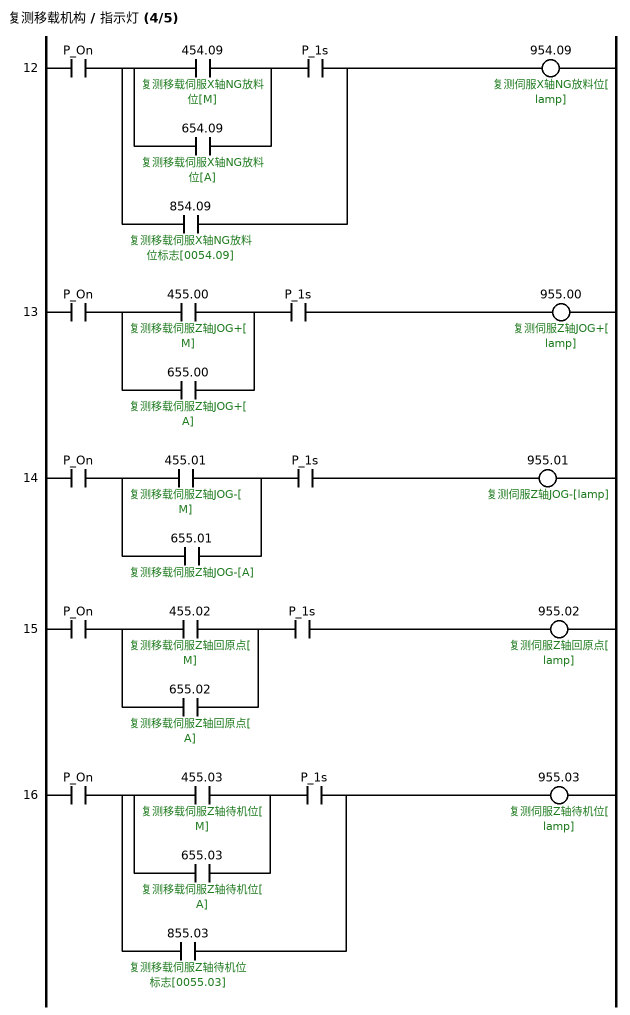
; [picture p576: 复测移载机构 / 指示灯, rungs 12-16]
; rung 12
LD P_On
LD 454.09  ; 复测移载伺服X轴NG放料位[M]
OR 654.09  ; 复测移载伺服X轴NG放料位[A]
AND P_1s
OR 854.09  ; 复测移载伺服X轴NG放料位标志[0054.09]
ANDLD
OUT 954.09  ; 复测伺服X轴NG放料位[lamp]
; rung 13
LD P_On
LD 455.00  ; 复测移载伺服Z轴JOG+[M]
OR 655.00  ; 复测移载伺服Z轴JOG+[A]
ANDLD
AND P_1s
OUT 955.00  ; 复测伺服Z轴JOG+[lamp]
; rung 14
LD P_On
LD 455.01  ; 复测移载伺服Z轴JOG-[M]
OR 655.01  ; 复测移载伺服Z轴JOG-[A]
ANDLD
AND P_1s
OUT 955.01  ; 复测伺服Z轴JOG-[lamp]
; rung 15
LD P_On
LD 455.02  ; 复测移载伺服Z轴回原点[M]
OR 655.02  ; 复测移载伺服Z轴回原点[A]
ANDLD
AND P_1s
OUT 955.02  ; 复测伺服Z轴回原点[lamp]
; rung 16
LD P_On
LD 455.03  ; 复测移载伺服Z轴待机位[M]
OR 655.03  ; 复测移载伺服Z轴待机位[A]
AND P_1s
OR 855.03  ; 复测移载伺服Z轴待机位标志[0055.03]
ANDLD
OUT 955.03  ; 复测伺服Z轴待机位[lamp]

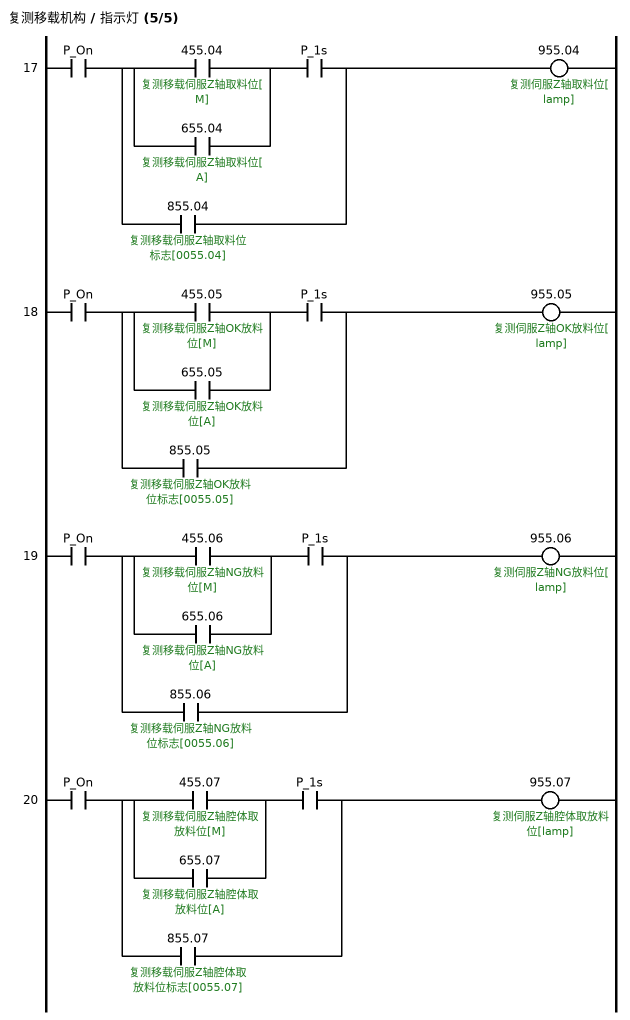
; rung 17
LD P_On
LD 455.04  ; 复测移载伺服Z轴取料位[M]
OR 655.04  ; 复测移载伺服Z轴取料位[A]
AND P_1s
OR 855.04  ; 复测移载伺服Z轴取料位标志[0055.04]
ANDLD
OUT 955.04  ; 复测伺服Z轴取料位[lamp]
; rung 18
LD P_On
LD 455.05  ; 复测移载伺服Z轴OK放料位[M]
OR 655.05  ; 复测移载伺服Z轴OK放料位[A]
AND P_1s
OR 855.05  ; 复测移载伺服Z轴OK放料位标志[0055.05]
ANDLD
OUT 955.05  ; 复测伺服Z轴OK放料位[lamp]
; rung 19
LD P_On
LD 455.06  ; 复测移载伺服Z轴NG放料位[M]
OR 655.06  ; 复测移载伺服Z轴NG放料位[A]
AND P_1s
OR 855.06  ; 复测移载伺服Z轴NG放料位标志[0055.06]
ANDLD
OUT 955.06  ; 复测伺服Z轴NG放料位[lamp]
; rung 20
LD P_On
LD 455.07  ; 复测移载伺服Z轴腔体取放料位[M]
OR 655.07  ; 复测移载伺服Z轴腔体取放料位[A]
AND P_1s
OR 855.07  ; 复测移载伺服Z轴腔体取放料位标志[0055.07]
ANDLD
OUT 955.07  ; 复测伺服Z轴腔体取放料位[lamp]

### Section 外部输出

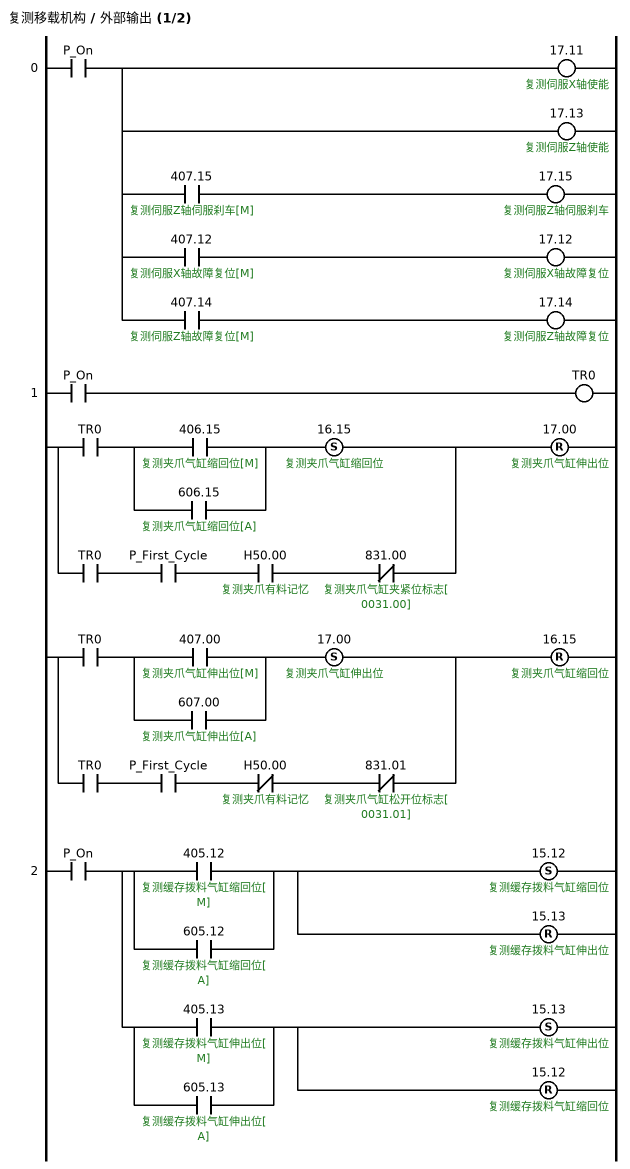
; rung 0
LD P_On
OUT TR0
OUT 17.11  ; 复测伺服X轴使能
OUT 17.13  ; 复测伺服Z轴使能
AND 407.15  ; 复测伺服Z轴伺服刹车[M]
OUT 17.15  ; 复测伺服Z轴伺服刹车
LD TR0
AND 407.12  ; 复测伺服X轴故障复位[M]
OUT 17.12  ; 复测伺服X轴故障复位
LD TR0
AND 407.14  ; 复测伺服Z轴故障复位[M]
OUT 17.14  ; 复测伺服Z轴故障复位
; rung 1
LD P_On
OUT TR0
LD 406.15  ; 复测夹爪气缸缩回位[M]
OR 606.15  ; 复测夹爪气缸缩回位[A]
ANDLD
SET 16.15  ; 复测夹爪气缸缩回位
LD TR0
AND P_First_Cycle
AND H50.00  ; 复测夹爪有料记忆
ANDNOT 831.00  ; 复测夹爪气缸夹紧位标志[0031.00]
ORLD
RSET 17.00  ; 复测夹爪气缸伸出位
LD TR0
LD 407.00  ; 复测夹爪气缸伸出位[M]
OR 607.00  ; 复测夹爪气缸伸出位[A]
ANDLD
SET 17.00  ; 复测夹爪气缸伸出位
LD TR0
AND P_First_Cycle
ANDNOT H50.00  ; 复测夹爪有料记忆
ANDNOT 831.01  ; 复测夹爪气缸松开位标志[0031.01]
ORLD
RSET 16.15  ; 复测夹爪气缸缩回位
; rung 2
LD P_On
OUT TR0
LD 405.12  ; 复测缓存拨料气缸缩回位[M]
OR 605.12  ; 复测缓存拨料气缸缩回位[A]
ANDLD
SET 15.12  ; 复测缓存拨料气缸缩回位
RSET 15.13  ; 复测缓存拨料气缸伸出位
LD TR0
LD 405.13  ; 复测缓存拨料气缸伸出位[M]
OR 605.13  ; 复测缓存拨料气缸伸出位[A]
ANDLD
SET 15.13  ; 复测缓存拨料气缸伸出位
RSET 15.12  ; 复测缓存拨料气缸缩回位

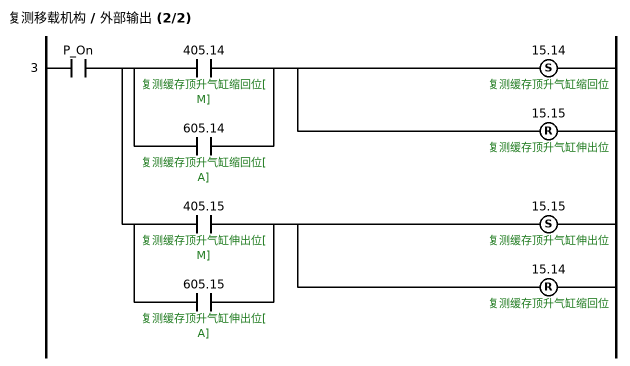
; rung 3
LD P_On
OUT TR0
LD 405.14  ; 复测缓存顶升气缸缩回位[M]
OR 605.14  ; 复测缓存顶升气缸缩回位[A]
ANDLD
SET 15.14  ; 复测缓存顶升气缸缩回位
RSET 15.15  ; 复测缓存顶升气缸伸出位
LD TR0
LD 405.15  ; 复测缓存顶升气缸伸出位[M]
OR 605.15  ; 复测缓存顶升气缸伸出位[A]
ANDLD
SET 15.15  ; 复测缓存顶升气缸伸出位
RSET 15.14  ; 复测缓存顶升气缸缩回位

### Section END
; rung 0
END(001)

## Program 复测腔体机构 (cyclic task 7)

### Section Main

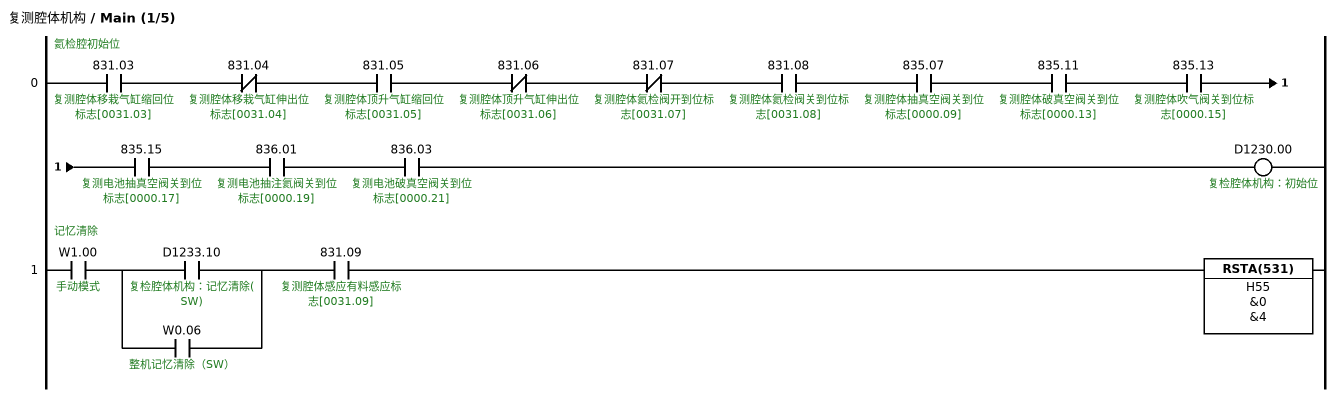
; rung 0: 氦检腔初始位
LD 831.03  ; 复测腔体移栽气缸缩回位标志[0031.03]
ANDNOT 831.04  ; 复测腔体移栽气缸伸出位标志[0031.04]
AND 831.05  ; 复测腔体顶升气缸缩回位标志[0031.05]
ANDNOT 831.06  ; 复测腔体顶升气缸伸出位标志[0031.06]
ANDNOT 831.07  ; 复测腔体氦检阀开到位标志[0031.07]
AND 831.08  ; 复测腔体氦检阀关到位标志[0031.08]
AND 835.07  ; 复测腔体抽真空阀关到位标志[0000.09]
AND 835.11  ; 复测腔体破真空阀关到位标志[0000.13]
AND 835.13  ; 复测腔体吹气阀关到位标志[0000.15]
AND 835.15  ; 复测电池抽真空阀关到位标志[0000.17]
AND 836.01  ; 复测电池抽注氦阀关到位标志[0000.19]
AND 836.03  ; 复测电池破真空阀关到位标志[0000.21]
OUT D1230.00  ; 复检腔体机构：初始位
; rung 1: 记忆清除
LD W1.00  ; 手动模式
LD D1233.10  ; 复检腔体机构：记忆清除(SW)
OR W0.06  ; 整机记忆清除（SW）
ANDLD
AND 831.09  ; 复测腔体感应有料感应标志[0031.09]
RSTA(531) H55 &0 &4

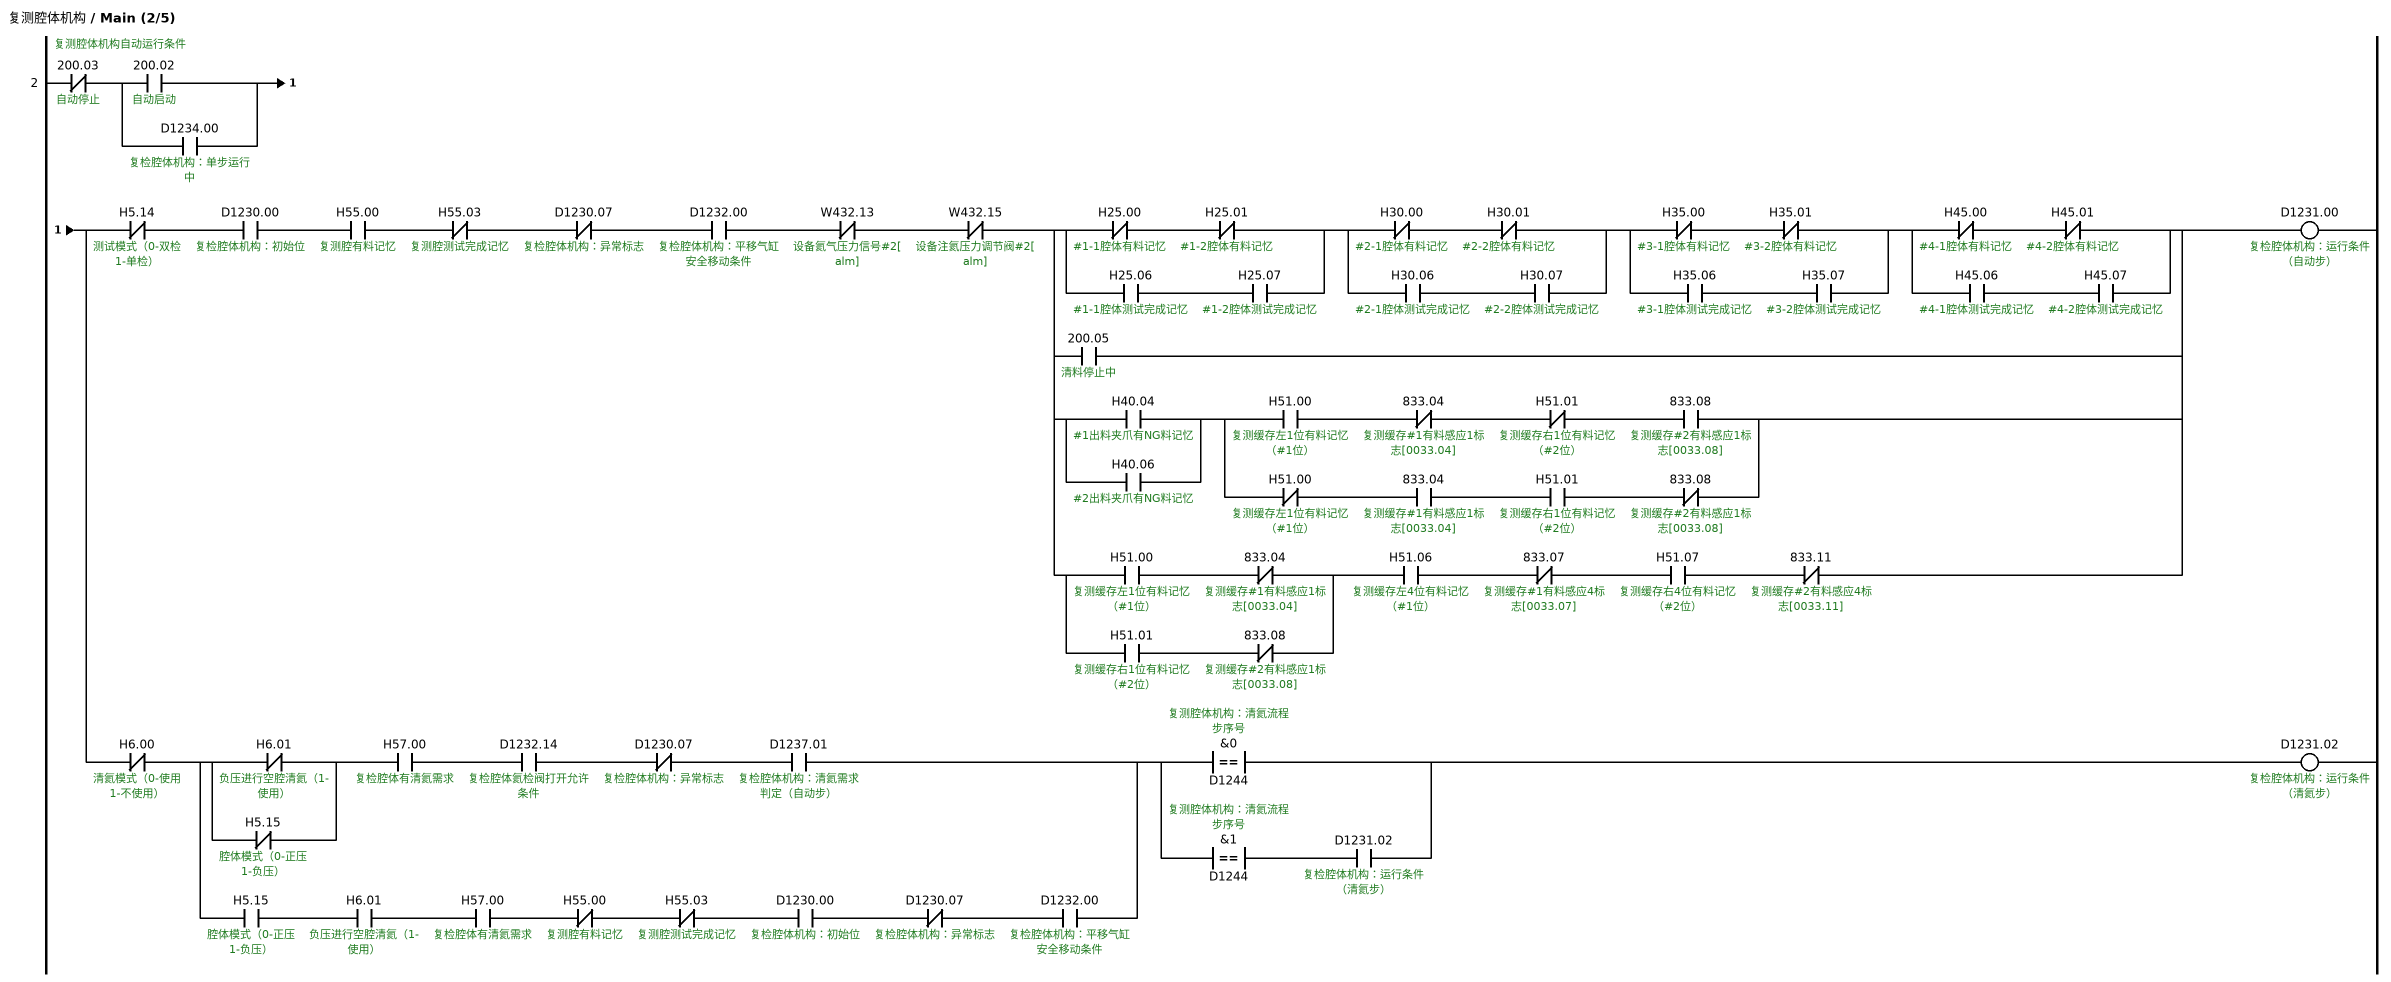
; rung 2: 复测腔体机构自动运行条件
LDNOT 200.03  ; 自动停止
LD 200.02  ; 自动启动
OR D1234.00  ; 复检腔体机构：单步运行中
ANDLD
OUT TR0
ANDNOT H5.14  ; 测试模式（0-双检 1-单检）
AND D1230.00  ; 复检腔体机构：初始位
AND H55.00  ; 复测腔有料记忆
ANDNOT H55.03  ; 复测腔测试完成记忆
ANDNOT D1230.07  ; 复检腔体机构：异常标志
AND D1232.00  ; 复检腔体机构：平移气缸安全移动条件
ANDNOT W432.13  ; 设备氦气压力信号#2[alm]
ANDNOT W432.15  ; 设备注氦压力调节阀#2[alm]
LDNOT H25.00  ; #1-1腔体有料记忆
ANDNOT H25.01  ; #1-2腔体有料记忆
LD H25.06  ; #1-1腔体测试完成记忆
AND H25.07  ; #1-2腔体测试完成记忆
ORLD
LDNOT H30.00  ; #2-1腔体有料记忆
ANDNOT H30.01  ; #2-2腔体有料记忆
LD H30.06  ; #2-1腔体测试完成记忆
AND H30.07  ; #2-2腔体测试完成记忆
ORLD
ANDLD
LDNOT H35.00  ; #3-1腔体有料记忆
ANDNOT H35.01  ; #3-2腔体有料记忆
LD H35.06  ; #3-1腔体测试完成记忆
AND H35.07  ; #3-2腔体测试完成记忆
ORLD
ANDLD
LDNOT H45.00  ; #4-1腔体有料记忆
ANDNOT H45.01  ; #4-2腔体有料记忆
LD H45.06  ; #4-1腔体测试完成记忆
AND H45.07  ; #4-2腔体测试完成记忆
ORLD
ANDLD
OR 200.05  ; 清料停止中
LD H40.04  ; #1出料夹爪有NG料记忆
OR H40.06  ; #2出料夹爪有NG料记忆
LD H51.00  ; 复测缓存左1位有料记忆（#1位）  // 缓存第一位出现单料是需直接清掉，防止下次待测料无法进行单个放料
ANDNOT 833.04  ; 复测缓存#1有料感应1标志[0033.04]
ANDNOT H51.01  ; 复测缓存右1位有料记忆（#2位）
AND 833.08  ; 复测缓存#2有料感应1标志[0033.08]
LDNOT H51.00  ; 复测缓存左1位有料记忆（#1位）
AND 833.04  ; 复测缓存#1有料感应1标志[0033.04]
AND H51.01  ; 复测缓存右1位有料记忆（#2位）
ANDNOT 833.08  ; 复测缓存#2有料感应1标志[0033.08]
ORLD
ANDLD
ORLD
LD H51.00  ; 复测缓存左1位有料记忆（#1位）
ANDNOT 833.04  ; 复测缓存#1有料感应1标志[0033.04]
LD H51.01  ; 复测缓存右1位有料记忆（#2位）
ANDNOT 833.08  ; 复测缓存#2有料感应1标志[0033.08]
ORLD
AND H51.06  ; 复测缓存左4位有料记忆（#1位）
ANDNOT 833.07  ; 复测缓存#1有料感应4标志[0033.07]
AND H51.07  ; 复测缓存右4位有料记忆（#2位）
ANDNOT 833.11  ; 复测缓存#2有料感应4标志[0033.11]
ORLD
ANDLD
OUT D1231.00  ; 复检腔体机构：运行条件（自动步）
LD TR0
ANDNOT H6.00  ; 清氦模式（0-使用 1-不使用）
LDNOT H6.01  ; 负压进行空腔清氦（1-使用）
ORNOT H5.15  ; 腔体模式（0-正压 1-负压）
AND H57.00  ; 复检腔体有清氦需求
AND D1232.14  ; 复检腔体氦检阀打开允许条件
ANDNOT D1230.07  ; 复检腔体机构：异常标志
AND D1237.01  ; 复检腔体机构：清氦需求判定（自动步）
LD H5.15  ; 腔体模式（0-正压 1-负压）
AND H6.01  ; 负压进行空腔清氦（1-使用）
AND H57.00  ; 复检腔体有清氦需求
ANDNOT H55.00  ; 复测腔有料记忆
ANDNOT H55.03  ; 复测腔测试完成记忆
AND D1230.00  ; 复检腔体机构：初始位
ANDNOT D1230.07  ; 复检腔体机构：异常标志
AND D1232.00  ; 复检腔体机构：平移气缸安全移动条件
ORLD
ANDLD
LD=L(301) &0 D1244  ; 复测腔体机构：清氦流程步序号
LD=L(301) &1 D1244  ; 复测腔体机构：清氦流程步序号
AND D1231.02  ; 复检腔体机构：运行条件（清氦步）
ORLD
ANDLD
OUT D1231.02  ; 复检腔体机构：运行条件（清氦步）

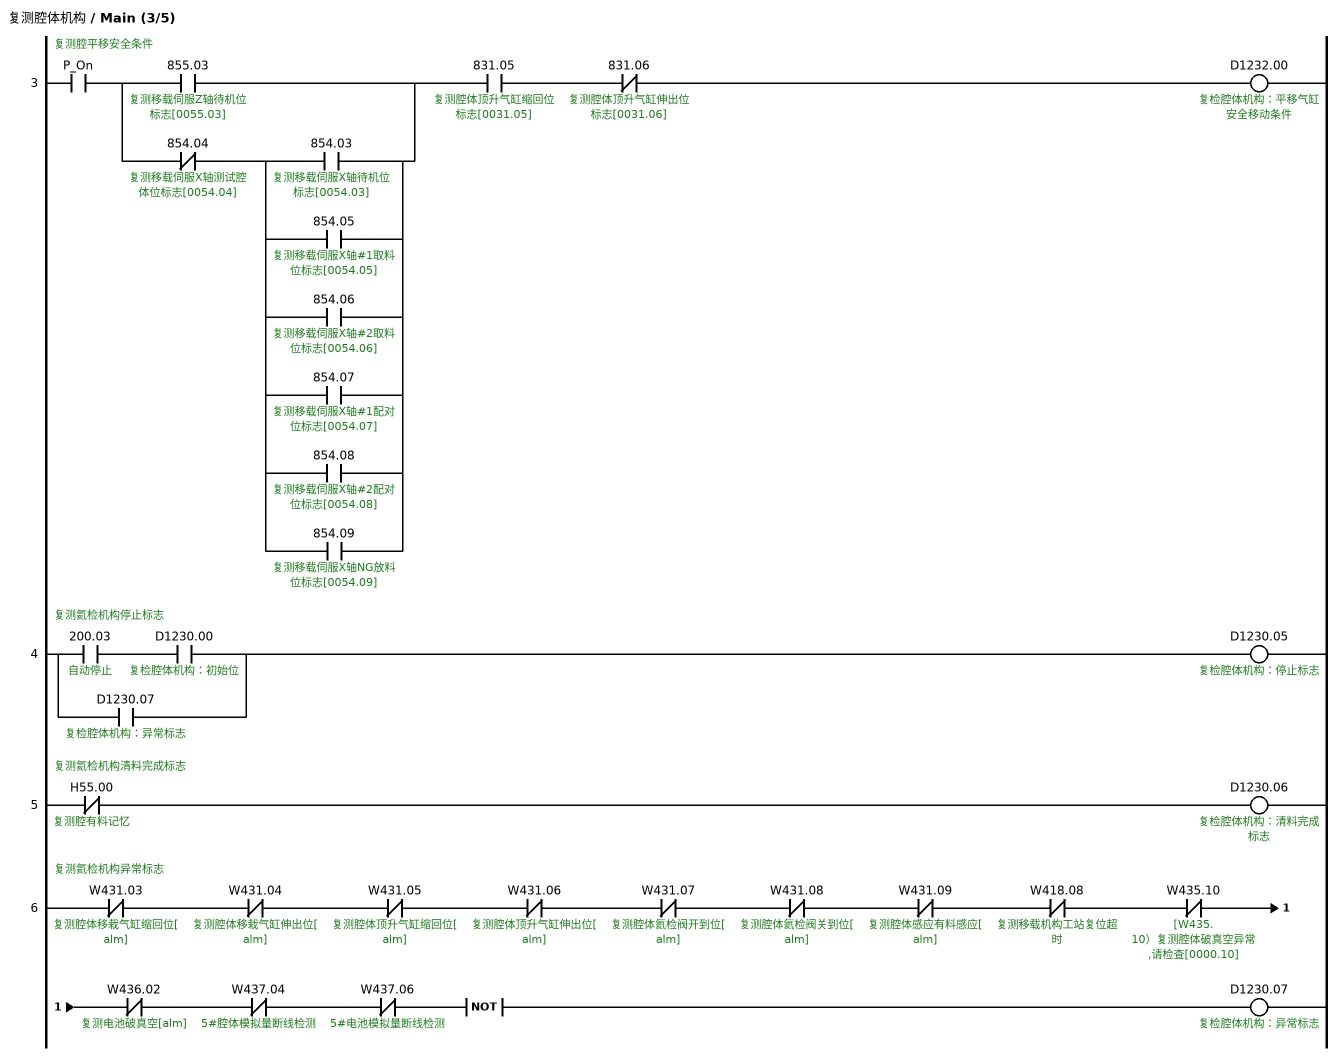
; rung 3: 复测腔平移安全条件
LD P_On
LD 855.03  ; 复测移载伺服Z轴待机位标志[0055.03]
LDNOT 854.04  ; 复测移载伺服X轴测试腔体位标志[0054.04]
LD 854.03  ; 复测移载伺服X轴待机位标志[0054.03]
OR 854.05  ; 复测移载伺服X轴#1取料位标志[0054.05]
OR 854.06  ; 复测移载伺服X轴#2取料位标志[0054.06]
OR 854.07  ; 复测移载伺服X轴#1配对位标志[0054.07]
OR 854.08  ; 复测移载伺服X轴#2配对位标志[0054.08]
OR 854.09  ; 复测移载伺服X轴NG放料位标志[0054.09]
ANDLD
ORLD
ANDLD
AND 831.05  ; 复测腔体顶升气缸缩回位标志[0031.05]
ANDNOT 831.06  ; 复测腔体顶升气缸伸出位标志[0031.06]
OUT D1232.00  ; 复检腔体机构：平移气缸安全移动条件
; rung 4: 复测氦检机构停止标志
LD 200.03  ; 自动停止
AND D1230.00  ; 复检腔体机构：初始位
OR D1230.07  ; 复检腔体机构：异常标志
OUT D1230.05  ; 复检腔体机构：停止标志
; rung 5: 复测氦检机构清料完成标志
LDNOT H55.00  ; 复测腔有料记忆
OUT D1230.06  ; 复检腔体机构：清料完成标志
; rung 6: 复测氦检机构异常标志
LDNOT W431.03  ; 复测腔体移栽气缸缩回位[alm]
ANDNOT W431.04  ; 复测腔体移栽气缸伸出位[alm]
ANDNOT W431.05  ; 复测腔体顶升气缸缩回位[alm]
ANDNOT W431.06  ; 复测腔体顶升气缸伸出位[alm]
ANDNOT W431.07  ; 复测腔体氦检阀开到位[alm]
ANDNOT W431.08  ; 复测腔体氦检阀关到位[alm]
ANDNOT W431.09  ; 复测腔体感应有料感应[alm]
ANDNOT W418.08  ; 复测移载机构工站复位超时
ANDNOT W435.10  ; [W435.10）复测腔体破真空异常,请检查[0000.10]
ANDNOT W436.02  ; 复测电池破真空[alm]
ANDNOT W437.04  ; 5#腔体模拟量断线检测
ANDNOT W437.06  ; 5#电池模拟量断线检测
NOT(520)
OUT D1230.07  ; 复检腔体机构：异常标志

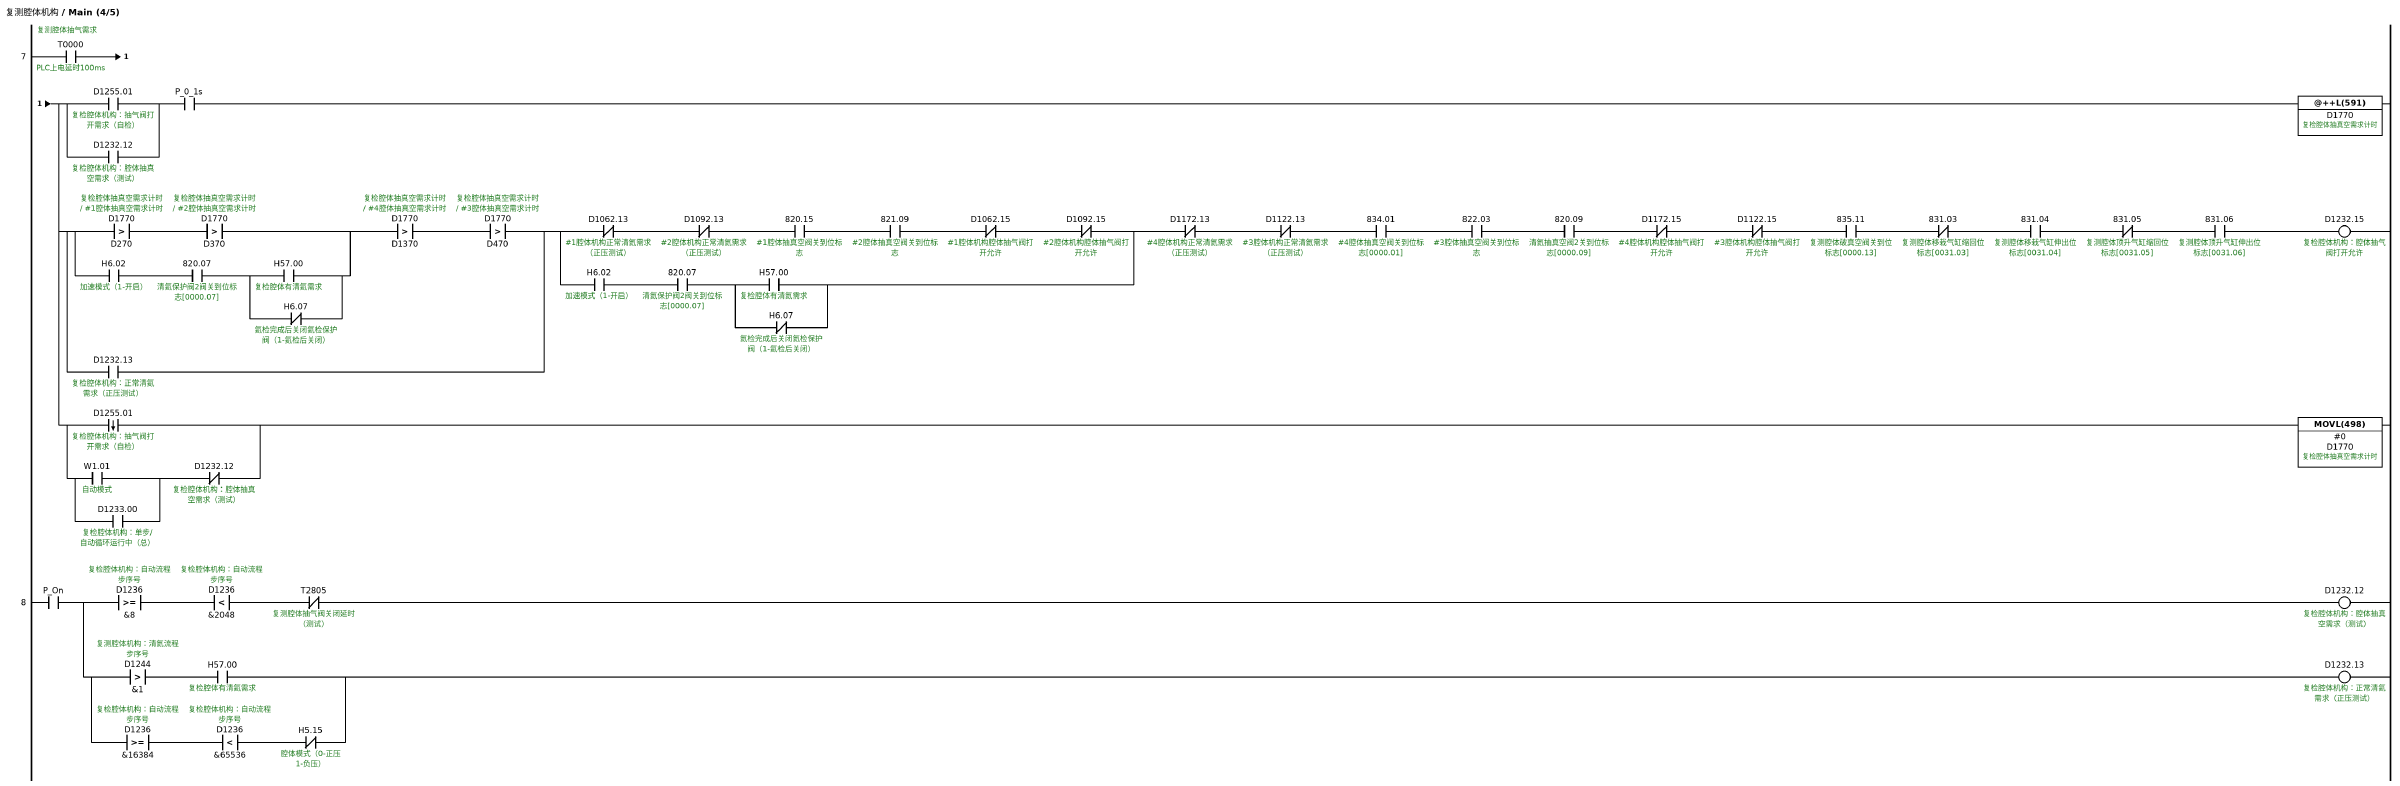
; rung 7: 复测腔体抽气需求
LD T0000  ; PLC上电延时100ms
OUT TR0
LD D1255.01  ; 复检腔体机构：抽气阀打开需求（自检）
OR D1232.12  ; 复检腔体机构：腔体抽真空需求（测试）
ANDLD
AND P_0_1s
@++L(591) D1770  ; 复检腔体抽真空需求计时
LD TR0
LD>L(321) D1770 D270  ; 复检腔体抽真空需求计时, #1腔体抽真空需求计时
AND>L(321) D1770 D370  ; 复检腔体抽真空需求计时, #2腔体抽真空需求计时
LD H6.02  ; 加速模式（1-开启）
AND 820.07  ; 清氦保护阀2阀关到位标志[0000.07]
LD H57.00  ; 复检腔体有清氦需求
ORNOT H6.07  ; 氦检完成后关闭氦检保护阀（1-氦检后关闭）
ANDLD
ORLD
AND>L(321) D1770 D1370  ; 复检腔体抽真空需求计时, #4腔体抽真空需求计时
AND>L(321) D1770 D470  ; 复检腔体抽真空需求计时, #3腔体抽真空需求计时
OR D1232.13  ; 复检腔体机构：正常清氦需求（正压测试）
ANDLD
LDNOT D1062.13  ; #1腔体机构正常清氦需求（正压测试）
ANDNOT D1092.13  ; #2腔体机构正常清氦需求（正压测试）
AND 820.15  ; #1腔体抽真空阀关到位标志
AND 821.09  ; #2腔体抽真空阀关到位标志
ANDNOT D1062.15  ; #1腔体机构腔体抽气阀打开允许
ANDNOT D1092.15  ; #2腔体机构腔体抽气阀打开允许
LD H6.02  ; 加速模式（1-开启）
AND 820.07  ; 清氦保护阀2阀关到位标志[0000.07]
LD H57.00  ; 复检腔体有清氦需求
ORNOT H6.07  ; 氦检完成后关闭氦检保护阀（1-氦检后关闭）
ANDLD
ORLD
ANDLD
ANDNOT D1172.13  ; #4腔体机构正常清氦需求（正压测试）
ANDNOT D1122.13  ; #3腔体机构正常清氦需求（正压测试）
AND 834.01  ; #4腔体抽真空阀关到位标志[0000.01]
AND 822.03  ; #3腔体抽真空阀关到位标志
AND 820.09  ; 清氦抽真空阀2关到位标志[0000.09]
ANDNOT D1172.15  ; #4腔体机构腔体抽气阀打开允许
ANDNOT D1122.15  ; #3腔体机构腔体抽气阀打开允许
AND 835.11  ; 复测腔体破真空阀关到位标志[0000.13]
ANDNOT 831.03  ; 复测腔体移栽气缸缩回位标志[0031.03]
AND 831.04  ; 复测腔体移栽气缸伸出位标志[0031.04]
ANDNOT 831.05  ; 复测腔体顶升气缸缩回位标志[0031.05]
AND 831.06  ; 复测腔体顶升气缸伸出位标志[0031.06]
OUT D1232.15  ; 复检腔体机构：腔体抽气阀打开允许
LD TR0
%LD D1255.01  ; 复检腔体机构：抽气阀打开需求（自检）
LD W1.01  ; 自动模式
OR D1233.00  ; 复检腔体机构：单步/自动循环运行中（总）
ANDNOT D1232.12  ; 复检腔体机构：腔体抽真空需求（测试）
ORLD
ANDLD
MOVL(498) #0 D1770  ; 复检腔体抽真空需求计时
; rung 8
LD P_On
OUT TR0
AND>=L(326) D1236 &8  ; 复检腔体机构：自动流程步序号
AND<L(311) D1236 &2048  ; 复检腔体机构：自动流程步序号
ANDNOT T2805  ; 复测腔体抽气阀关闭延时（测试）
OUT D1232.12  ; 复检腔体机构：腔体抽真空需求（测试）
LD TR0
LD>L(321) D1244 &1  ; 复测腔体机构：清氦流程步序号
AND H57.00  ; 复检腔体有清氦需求
LD>=L(326) D1236 &16384  ; 复检腔体机构：自动流程步序号
AND<L(311) D1236 &65536  ; 复检腔体机构：自动流程步序号
ANDNOT H5.15  ; 腔体模式（0-正压 1-负压）
ORLD
ANDLD
OUT D1232.13  ; 复检腔体机构：正常清氦需求（正压测试）

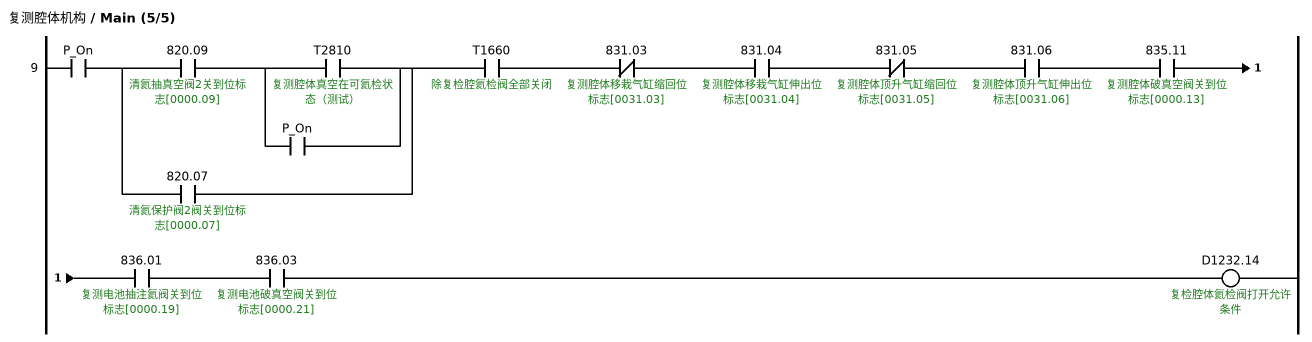
; rung 9
LD P_On
LD 820.09  ; 清氦抽真空阀2关到位标志[0000.09]
LD T2810  ; 复测腔体真空在可氦检状态（测试）
OR P_On
ANDLD
OR 820.07  ; 清氦保护阀2阀关到位标志[0000.07]
ANDLD
AND T1660  ; 除复检腔氦检阀全部关闭
ANDNOT 831.03  ; 复测腔体移栽气缸缩回位标志[0031.03]
AND 831.04  ; 复测腔体移栽气缸伸出位标志[0031.04]
ANDNOT 831.05  ; 复测腔体顶升气缸缩回位标志[0031.05]
AND 831.06  ; 复测腔体顶升气缸伸出位标志[0031.06]
AND 835.11  ; 复测腔体破真空阀关到位标志[0000.13]
AND 836.01  ; 复测电池抽注氦阀关到位标志[0000.19]
AND 836.03  ; 复测电池破真空阀关到位标志[0000.21]
OUT D1232.14  ; 复检腔体氦检阀打开允许条件

### Section 复测腔自动

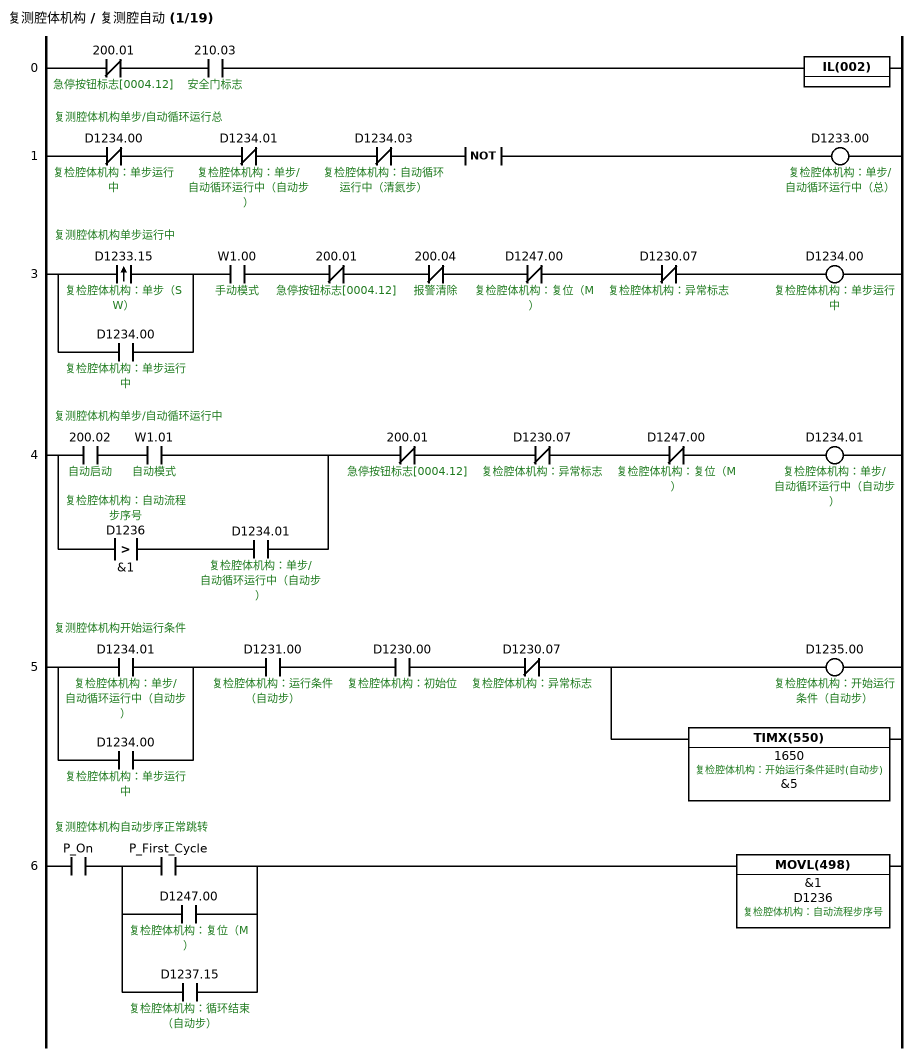
; rung 0
LDNOT 200.01  ; 急停按钮标志[0004.12]
AND 210.03  ; 安全门标志
IL(002)
; rung 1: 复测腔体机构单步/自动循环运行总
LDNOT D1234.00  ; 复检腔体机构：单步运行中
ANDNOT D1234.01  ; 复检腔体机构：单步/自动循环运行中（自动步）
ANDNOT D1234.03  ; 复检腔体机构：自动循环运行中（清氦步）
NOT(520)
OUT D1233.00  ; 复检腔体机构：单步/自动循环运行中（总）
; rung 2: ******************************* / 自动双检步序 / *******************************
; rung 3: 复测腔体机构单步运行中
@LD D1233.15  ; 复检腔体机构：单步（SW）
OR D1234.00  ; 复检腔体机构：单步运行中
AND W1.00  ; 手动模式
ANDNOT 200.01  ; 急停按钮标志[0004.12]
ANDNOT 200.04  ; 报警清除
ANDNOT D1247.00  ; 复检腔体机构：复位（M）
ANDNOT D1230.07  ; 复检腔体机构：异常标志
OUT D1234.00  ; 复检腔体机构：单步运行中
; rung 4: 复测腔体机构单步/自动循环运行中
LD 200.02  ; 自动启动
AND W1.01  ; 自动模式
LD>L(321) D1236 &1  ; 复检腔体机构：自动流程步序号
AND D1234.01  ; 复检腔体机构：单步/自动循环运行中（自动步）
ORLD
ANDNOT 200.01  ; 急停按钮标志[0004.12]
ANDNOT D1230.07  ; 复检腔体机构：异常标志
ANDNOT D1247.00  ; 复检腔体机构：复位（M）
OUT D1234.01  ; 复检腔体机构：单步/自动循环运行中（自动步）
; rung 5: 复测腔体机构开始运行条件
LD D1234.01  ; 复检腔体机构：单步/自动循环运行中（自动步）
OR D1234.00  ; 复检腔体机构：单步运行中
AND D1231.00  ; 复检腔体机构：运行条件（自动步）
AND D1230.00  ; 复检腔体机构：初始位
ANDNOT D1230.07  ; 复检腔体机构：异常标志
OUT D1235.00  ; 复检腔体机构：开始运行条件（自动步）
TIMX(550) 1650 &5  ; 复检腔体机构：开始运行条件延时(自动步)
; rung 6: 复测腔体机构自动步序正常跳转
LD P_On
LD P_First_Cycle
OR D1247.00  ; 复检腔体机构：复位（M）
OR D1237.15  ; 复检腔体机构：循环结束（自动步）
ANDLD
MOVL(498) &1 D1236  ; 复检腔体机构：自动流程步序号

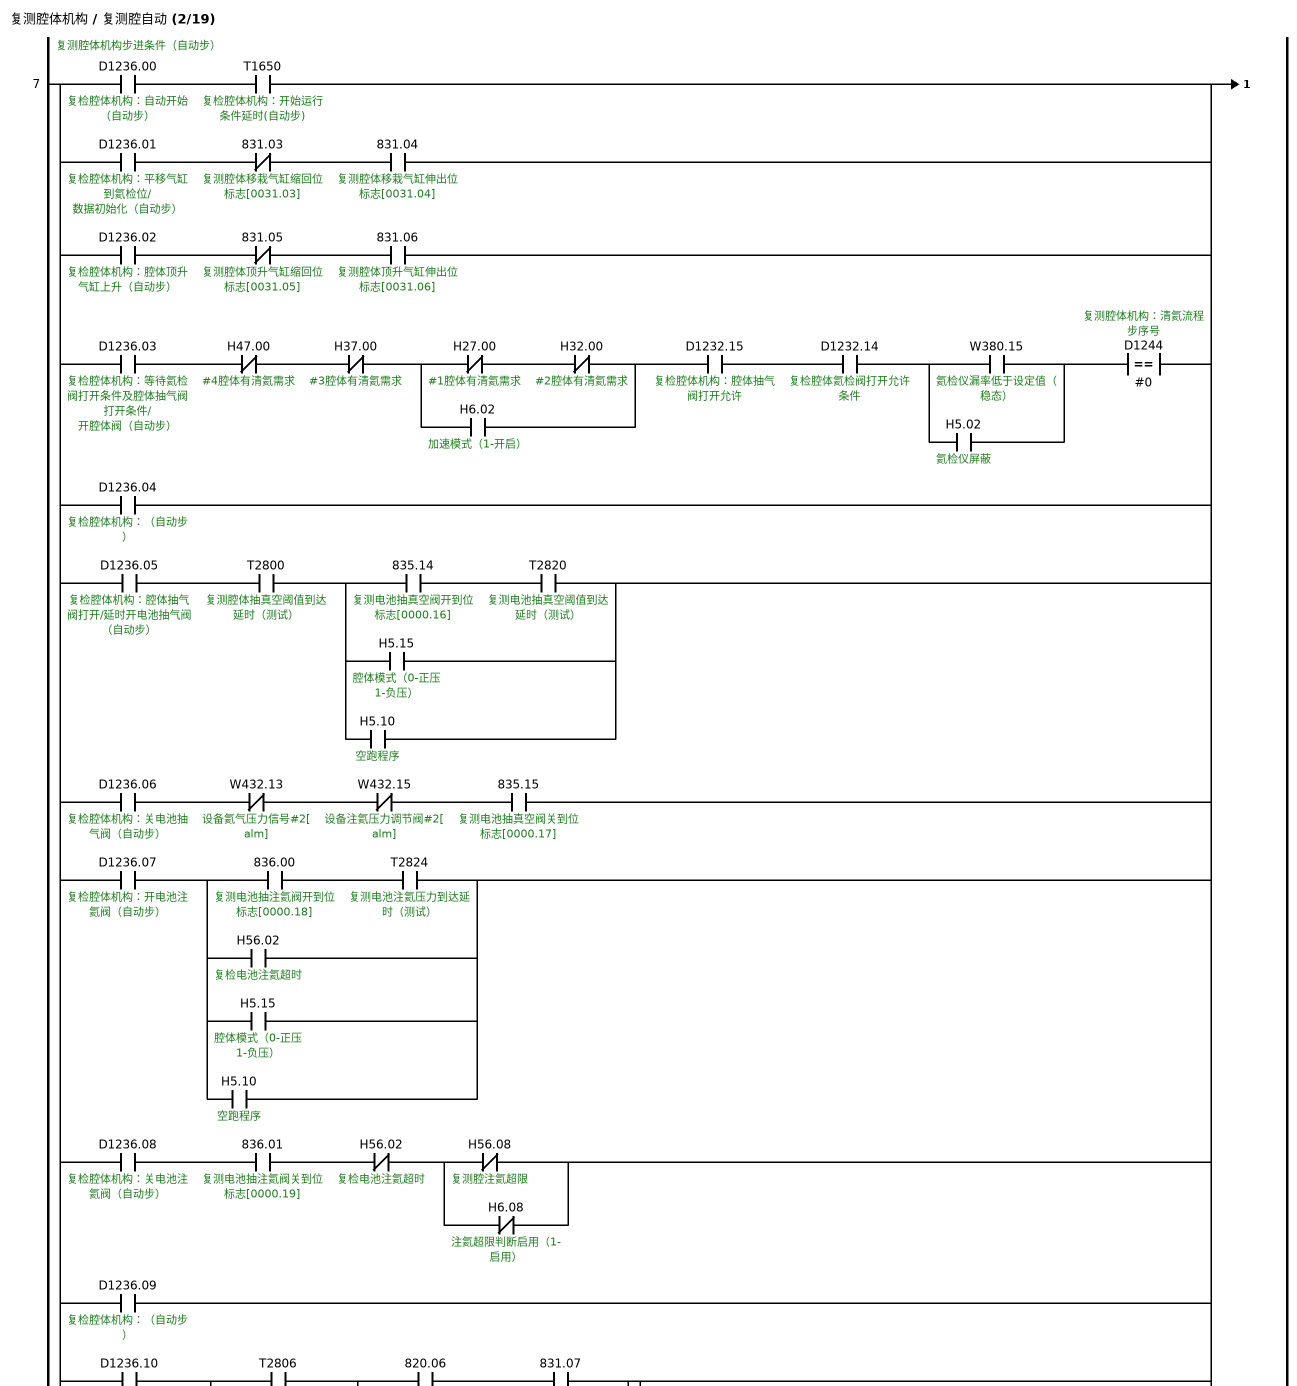

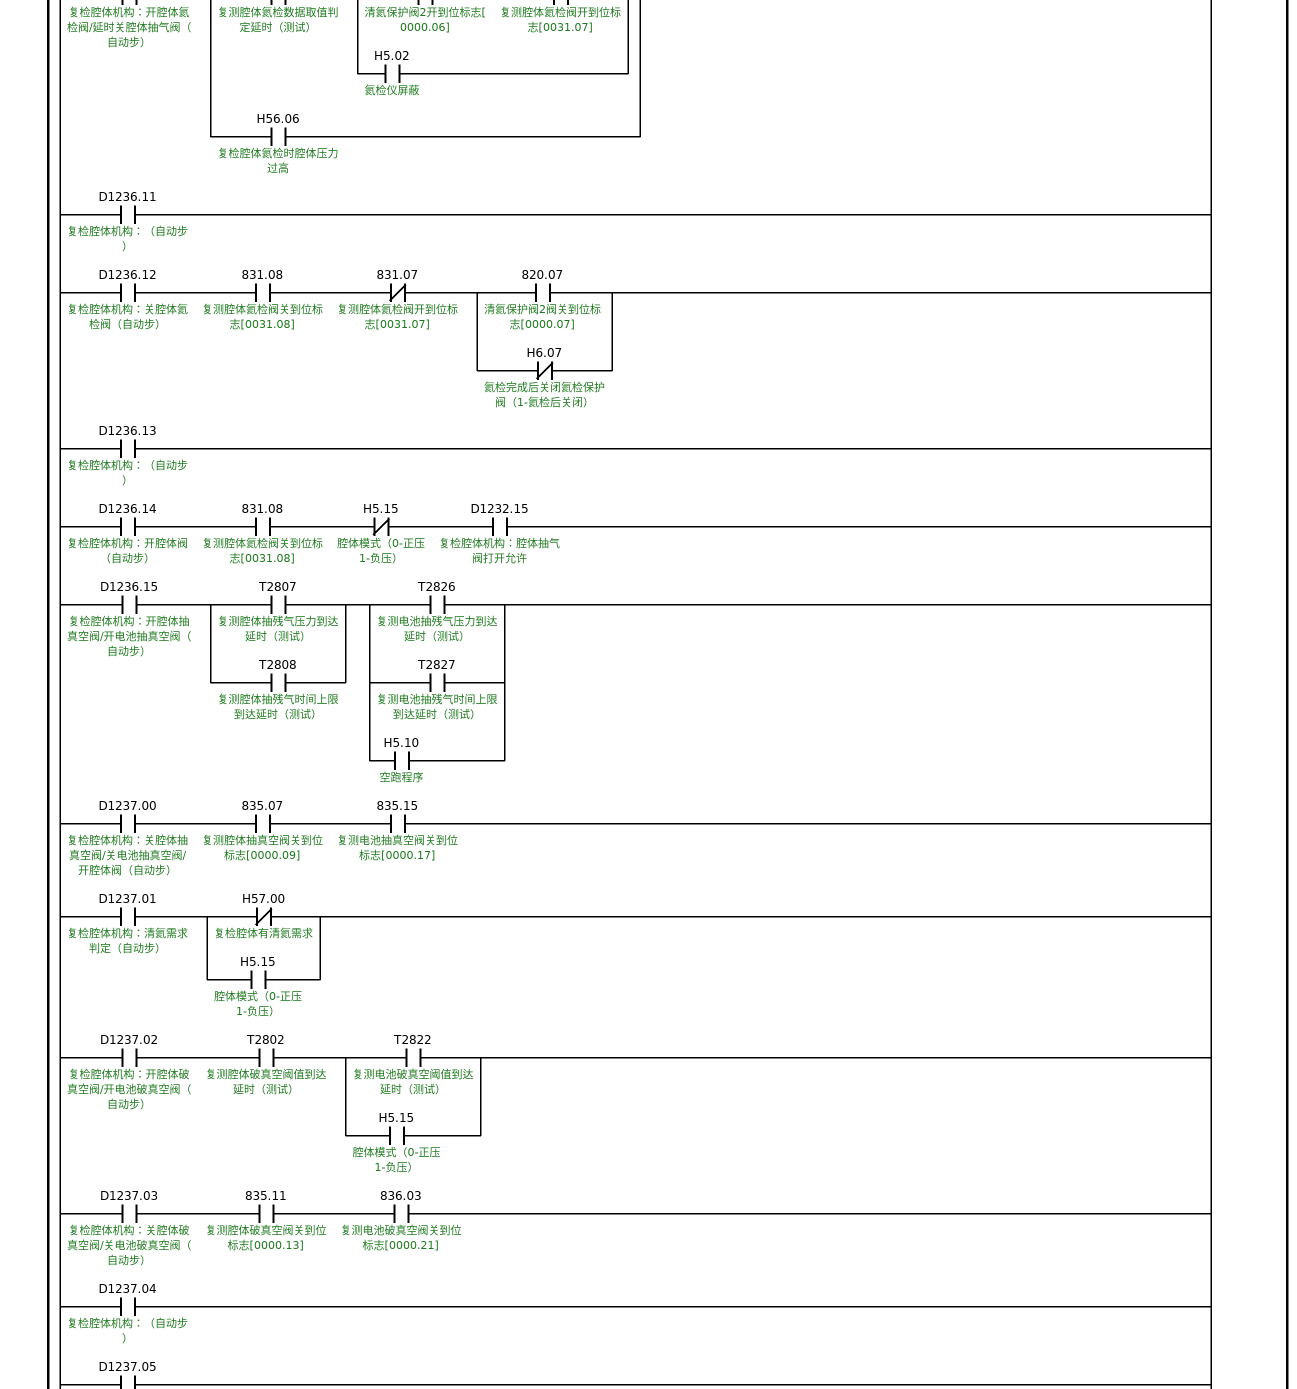

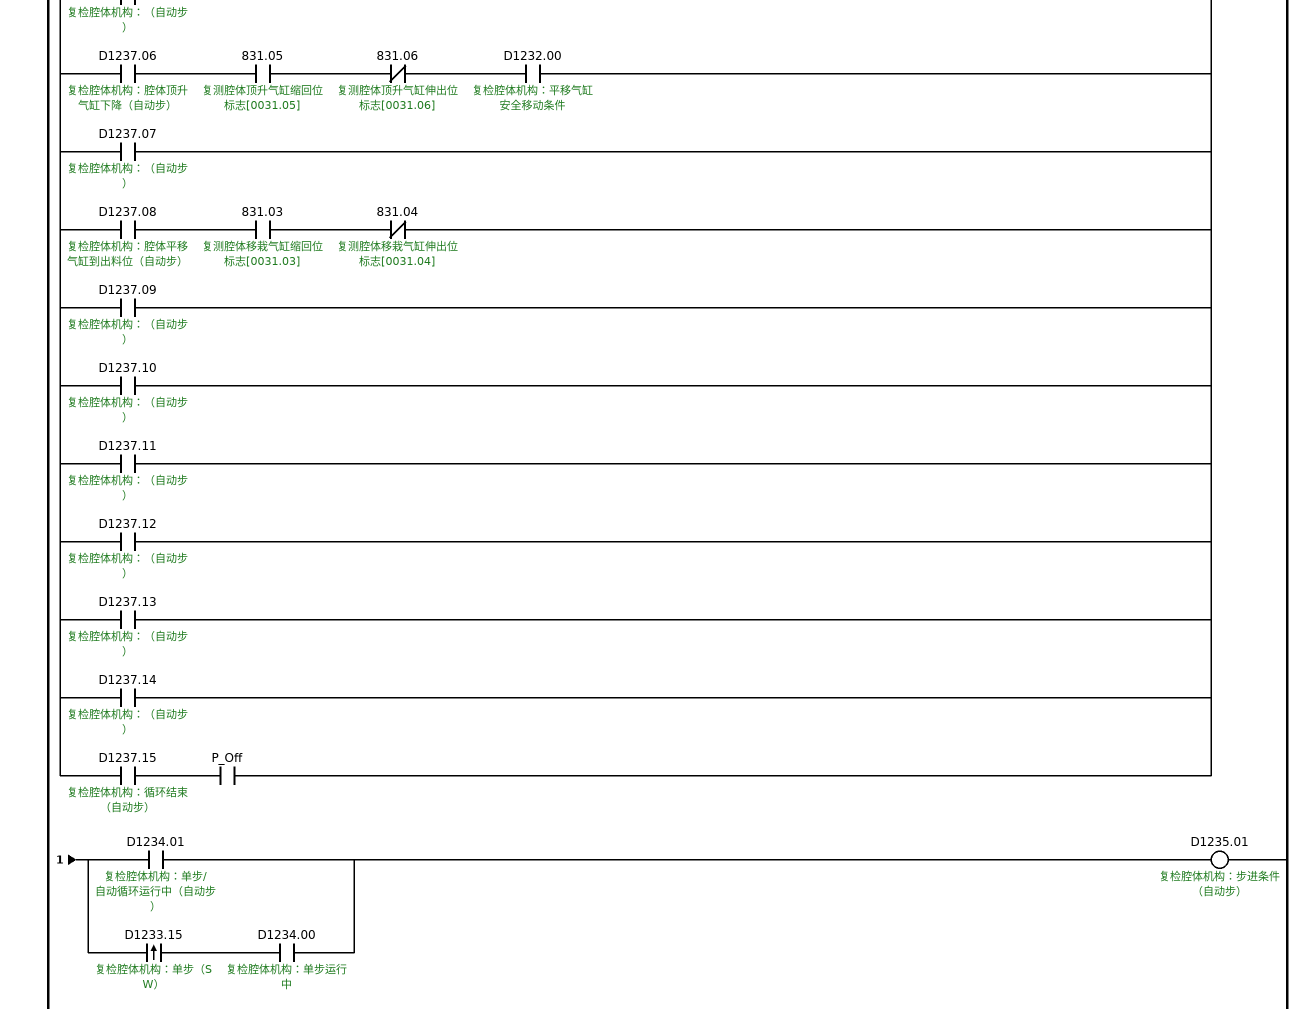
; rung 7: 复测腔体机构步进条件（自动步）
LD D1236.00  ; 复检腔体机构：自动开始（自动步）
AND T1650  ; 复检腔体机构：开始运行条件延时(自动步)
LD D1236.01  ; 复检腔体机构：平移气缸到氦检位/数据初始化（自动步）
ANDNOT 831.03  ; 复测腔体移栽气缸缩回位标志[0031.03]
AND 831.04  ; 复测腔体移栽气缸伸出位标志[0031.04]
ORLD
LD D1236.02  ; 复检腔体机构：腔体顶升气缸上升（自动步）
ANDNOT 831.05  ; 复测腔体顶升气缸缩回位标志[0031.05]
AND 831.06  ; 复测腔体顶升气缸伸出位标志[0031.06]
ORLD
LD D1236.03  ; 复检腔体机构：等待氦检阀打开条件及腔体抽气阀打开条件/开腔体阀（自动步）
ANDNOT H47.00  ; #4腔体有清氦需求
ANDNOT H37.00  ; #3腔体有清氦需求
LDNOT H27.00  ; #1腔体有清氦需求
ANDNOT H32.00  ; #2腔体有清氦需求
OR H6.02  ; 加速模式（1-开启）
ANDLD
AND D1232.15  ; 复检腔体机构：腔体抽气阀打开允许
AND D1232.14  ; 复检腔体氦检阀打开允许条件
LD W380.15  ; 氦检仪漏率低于设定值（稳态）
OR H5.02  ; 氦检仪屏蔽
ANDLD
AND=L(301) D1244 #0  ; 复测腔体机构：清氦流程步序号
ORLD
OR D1236.04  ; 复检腔体机构：（自动步）
LD D1236.05  ; 复检腔体机构：腔体抽气阀打开/延时开电池抽气阀（自动步）
AND T2800  ; 复测腔体抽真空阈值到达延时（测试）
LD 835.14  ; 复测电池抽真空阀开到位标志[0000.16]
AND T2820  ; 复测电池抽真空阈值到达延时（测试）
OR H5.15  ; 腔体模式（0-正压 1-负压）
OR H5.10  ; 空跑程序
ANDLD
ORLD
LD D1236.06  ; 复检腔体机构：关电池抽气阀（自动步）
ANDNOT W432.13  ; 设备氦气压力信号#2[alm]
ANDNOT W432.15  ; 设备注氦压力调节阀#2[alm]
AND 835.15  ; 复测电池抽真空阀关到位标志[0000.17]
ORLD
LD D1236.07  ; 复检腔体机构：开电池注氦阀（自动步）
LD 836.00  ; 复测电池抽注氦阀开到位标志[0000.18]
AND T2824  ; 复测电池注氦压力到达延时（测试）
OR H56.02  ; 复检电池注氦超时
OR H5.15  ; 腔体模式（0-正压 1-负压）
OR H5.10  ; 空跑程序
ANDLD
ORLD
LD D1236.08  ; 复检腔体机构：关电池注氦阀（自动步）
AND 836.01  ; 复测电池抽注氦阀关到位标志[0000.19]
ANDNOT H56.02  ; 复检电池注氦超时
LDNOT H56.08  ; 复测腔注氦超限
ORNOT H6.08  ; 注氦超限判断启用（1-启用）
ANDLD
ORLD
OR D1236.09  ; 复检腔体机构：（自动步）
LD D1236.10  ; 复检腔体机构：开腔体氦检阀/延时关腔体抽气阀（自动步）
LD T2806  ; 复测腔体氦检数据取值判定延时（测试）
LD 820.06  ; 清氦保护阀2开到位标志[0000.06]
AND 831.07  ; 复测腔体氦检阀开到位标志[0031.07]
OR H5.02  ; 氦检仪屏蔽
ANDLD
OR H56.06  ; 复检腔体氦检时腔体压力过高
ANDLD
ORLD
OR D1236.11  ; 复检腔体机构：（自动步）
LD D1236.12  ; 复检腔体机构：关腔体氦检阀（自动步）
AND 831.08  ; 复测腔体氦检阀关到位标志[0031.08]
ANDNOT 831.07  ; 复测腔体氦检阀开到位标志[0031.07]
LD 820.07  ; 清氦保护阀2阀关到位标志[0000.07]
ORNOT H6.07  ; 氦检完成后关闭氦检保护阀（1-氦检后关闭）
ANDLD
ORLD
OR D1236.13  ; 复检腔体机构：（自动步）
LD D1236.14  ; 复检腔体机构：开腔体阀（自动步）  // 负压模式正常电池不进行抽真空，直接跳转
AND 831.08  ; 复测腔体氦检阀关到位标志[0031.08]
ANDNOT H5.15  ; 腔体模式（0-正压 1-负压）
AND D1232.15  ; 复检腔体机构：腔体抽气阀打开允许
ORLD
LD D1236.15  ; 复检腔体机构：开腔体抽真空阀/开电池抽真空阀（自动步）
LD T2807  ; 复测腔体抽残气压力到达延时（测试）
OR T2808  ; 复测腔体抽残气时间上限到达延时（测试）
ANDLD
LD T2826  ; 复测电池抽残气压力到达延时（测试）
OR T2827  ; 复测电池抽残气时间上限到达延时（测试）
OR H5.10  ; 空跑程序
ANDLD
ORLD
LD D1237.00  ; 复检腔体机构：关腔体抽真空阀/关电池抽真空阀/开腔体阀（自动步）
AND 835.07  ; 复测腔体抽真空阀关到位标志[0000.09]
AND 835.15  ; 复测电池抽真空阀关到位标志[0000.17]
ORLD
LD D1237.01  ; 复检腔体机构：清氦需求判定（自动步）
LDNOT H57.00  ; 复检腔体有清氦需求
OR H5.15  ; 腔体模式（0-正压 1-负压）
ANDLD
ORLD
LD D1237.02  ; 复检腔体机构：开腔体破真空阀/开电池破真空阀（自动步）
AND T2802  ; 复测腔体破真空阈值到达延时（测试）
LD T2822  ; 复测电池破真空阈值到达延时（测试）
OR H5.15  ; 腔体模式（0-正压 1-负压）
ANDLD
ORLD
LD D1237.03  ; 复检腔体机构：关腔体破真空阀/关电池破真空阀（自动步）
AND 835.11  ; 复测腔体破真空阀关到位标志[0000.13]
AND 836.03  ; 复测电池破真空阀关到位标志[0000.21]
ORLD
OR D1237.04  ; 复检腔体机构：（自动步）
OR D1237.05  ; 复检腔体机构：（自动步）
LD D1237.06  ; 复检腔体机构：腔体顶升气缸下降（自动步）
AND 831.05  ; 复测腔体顶升气缸缩回位标志[0031.05]
ANDNOT 831.06  ; 复测腔体顶升气缸伸出位标志[0031.06]
AND D1232.00  ; 复检腔体机构：平移气缸安全移动条件
ORLD
OR D1237.07  ; 复检腔体机构：（自动步）
LD D1237.08  ; 复检腔体机构：腔体平移气缸到出料位（自动步）
AND 831.03  ; 复测腔体移栽气缸缩回位标志[0031.03]
ANDNOT 831.04  ; 复测腔体移栽气缸伸出位标志[0031.04]
ORLD
OR D1237.09  ; 复检腔体机构：（自动步）
OR D1237.10  ; 复检腔体机构：（自动步）
OR D1237.11  ; 复检腔体机构：（自动步）
OR D1237.12  ; 复检腔体机构：（自动步）
OR D1237.13  ; 复检腔体机构：（自动步）
OR D1237.14  ; 复检腔体机构：（自动步）
LD D1237.15  ; 复检腔体机构：循环结束（自动步）
AND P_Off
ORLD
LD D1234.01  ; 复检腔体机构：单步/自动循环运行中（自动步）
@LD D1233.15  ; 复检腔体机构：单步（SW）
AND D1234.00  ; 复检腔体机构：单步运行中
ORLD
ANDLD
OUT D1235.01  ; 复检腔体机构：步进条件（自动步）

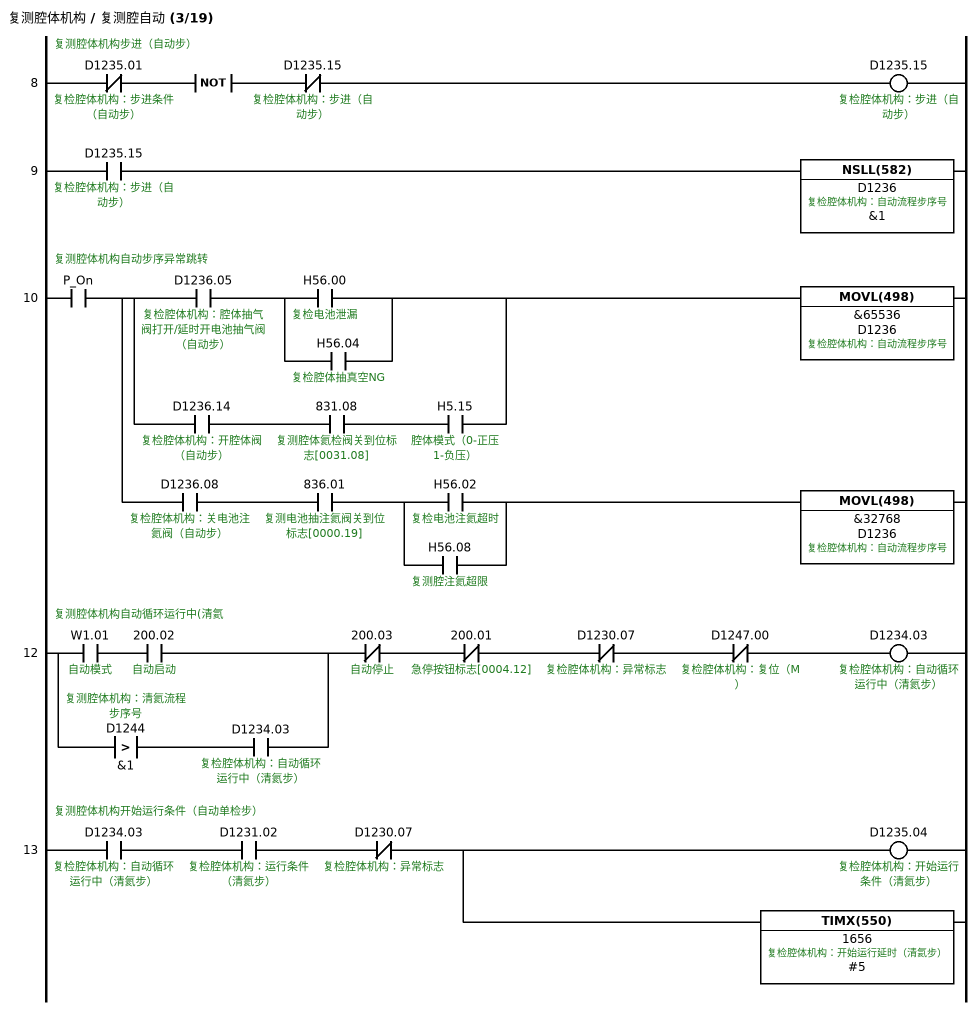
; rung 8: 复测腔体机构步进（自动步）
LDNOT D1235.01  ; 复检腔体机构：步进条件（自动步）
NOT(520)
ANDNOT D1235.15  ; 复检腔体机构：步进（自动步）
OUT D1235.15  ; 复检腔体机构：步进（自动步）
; rung 9
LD D1235.15  ; 复检腔体机构：步进（自动步）
NSLL(582) D1236 &1  ; 复检腔体机构：自动流程步序号
; rung 10: 复测腔体机构自动步序异常跳转
LD P_On
OUT TR0
LD D1236.05  ; 复检腔体机构：腔体抽气阀打开/延时开电池抽气阀（自动步）
LD H56.00  ; 复检电池泄漏
OR H56.04  ; 复检腔体抽真空NG
ANDLD
LD D1236.14  ; 复检腔体机构：开腔体阀（自动步）  // 负压模式不需要进行氦检后抽真空动作
AND 831.08  ; 复测腔体氦检阀关到位标志[0031.08]
AND H5.15  ; 腔体模式（0-正压 1-负压）
ORLD
ANDLD
MOVL(498) &65536 D1236  ; 复检腔体机构：自动流程步序号  // 出现腔体抽真空NG，电池抽真空NG，均跳转至自动步序D1067.0
LD TR0
AND D1236.08  ; 复检腔体机构：关电池注氦阀（自动步）
AND 836.01  ; 复测电池抽注氦阀关到位标志[0000.19]
LD H56.02  ; 复检电池注氦超时
OR H56.08  ; 复测腔注氦超限
ANDLD
MOVL(498) &32768 D1236  ; 复检腔体机构：自动流程步序号  // 电池注氦超时的情况，需跳转至d1236.15
; rung 11: ******************************* / 清氦步序 / *******************************
; rung 12: 复测腔体机构自动循环运行中(清氦
LD W1.01  ; 自动模式
AND 200.02  ; 自动启动
LD>L(321) D1244 &1  ; 复测腔体机构：清氦流程步序号
AND D1234.03  ; 复检腔体机构：自动循环运行中（清氦步）
ORLD
ANDNOT 200.03  ; 自动停止
ANDNOT 200.01  ; 急停按钮标志[0004.12]
ANDNOT D1230.07  ; 复检腔体机构：异常标志
ANDNOT D1247.00  ; 复检腔体机构：复位（M）
OUT D1234.03  ; 复检腔体机构：自动循环运行中（清氦步）
; rung 13: 复测腔体机构开始运行条件（自动单检步）
LD D1234.03  ; 复检腔体机构：自动循环运行中（清氦步）
AND D1231.02  ; 复检腔体机构：运行条件（清氦步）
ANDNOT D1230.07  ; 复检腔体机构：异常标志
OUT D1235.04  ; 复检腔体机构：开始运行条件（清氦步）
TIMX(550) 1656 #5  ; 复检腔体机构：开始运行延时（清氦步）

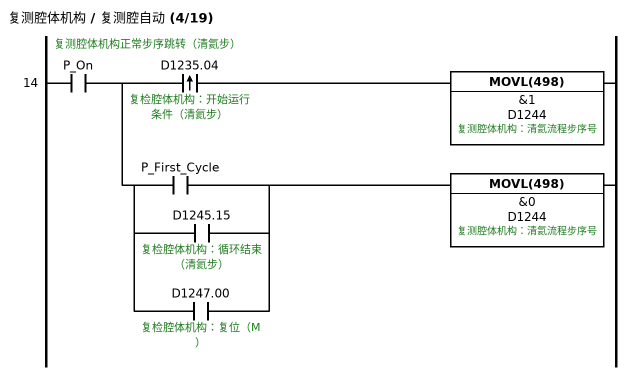
; rung 14: 复测腔体机构正常步序跳转（清氦步）
LD P_On
OUT TR0
@AND D1235.04  ; 复检腔体机构：开始运行条件（清氦步）
MOVL(498) &1 D1244  ; 复测腔体机构：清氦流程步序号
LD TR0
LD P_First_Cycle
OR D1245.15  ; 复检腔体机构：循环结束（清氦步）
OR D1247.00  ; 复检腔体机构：复位（M）
ANDLD
MOVL(498) &0 D1244  ; 复测腔体机构：清氦流程步序号

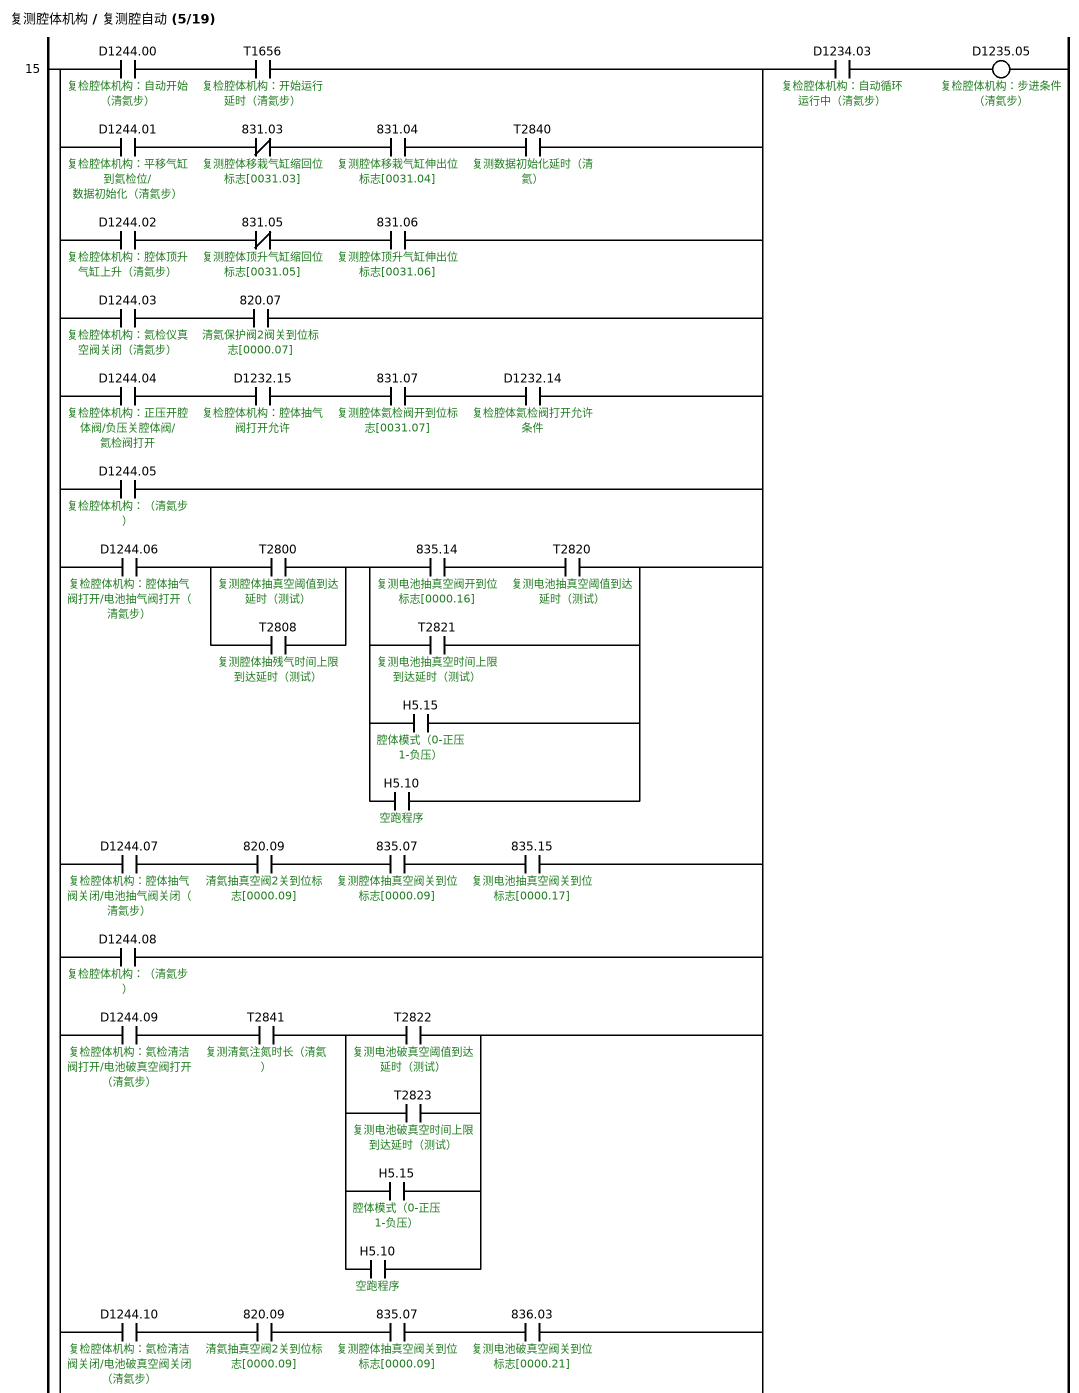

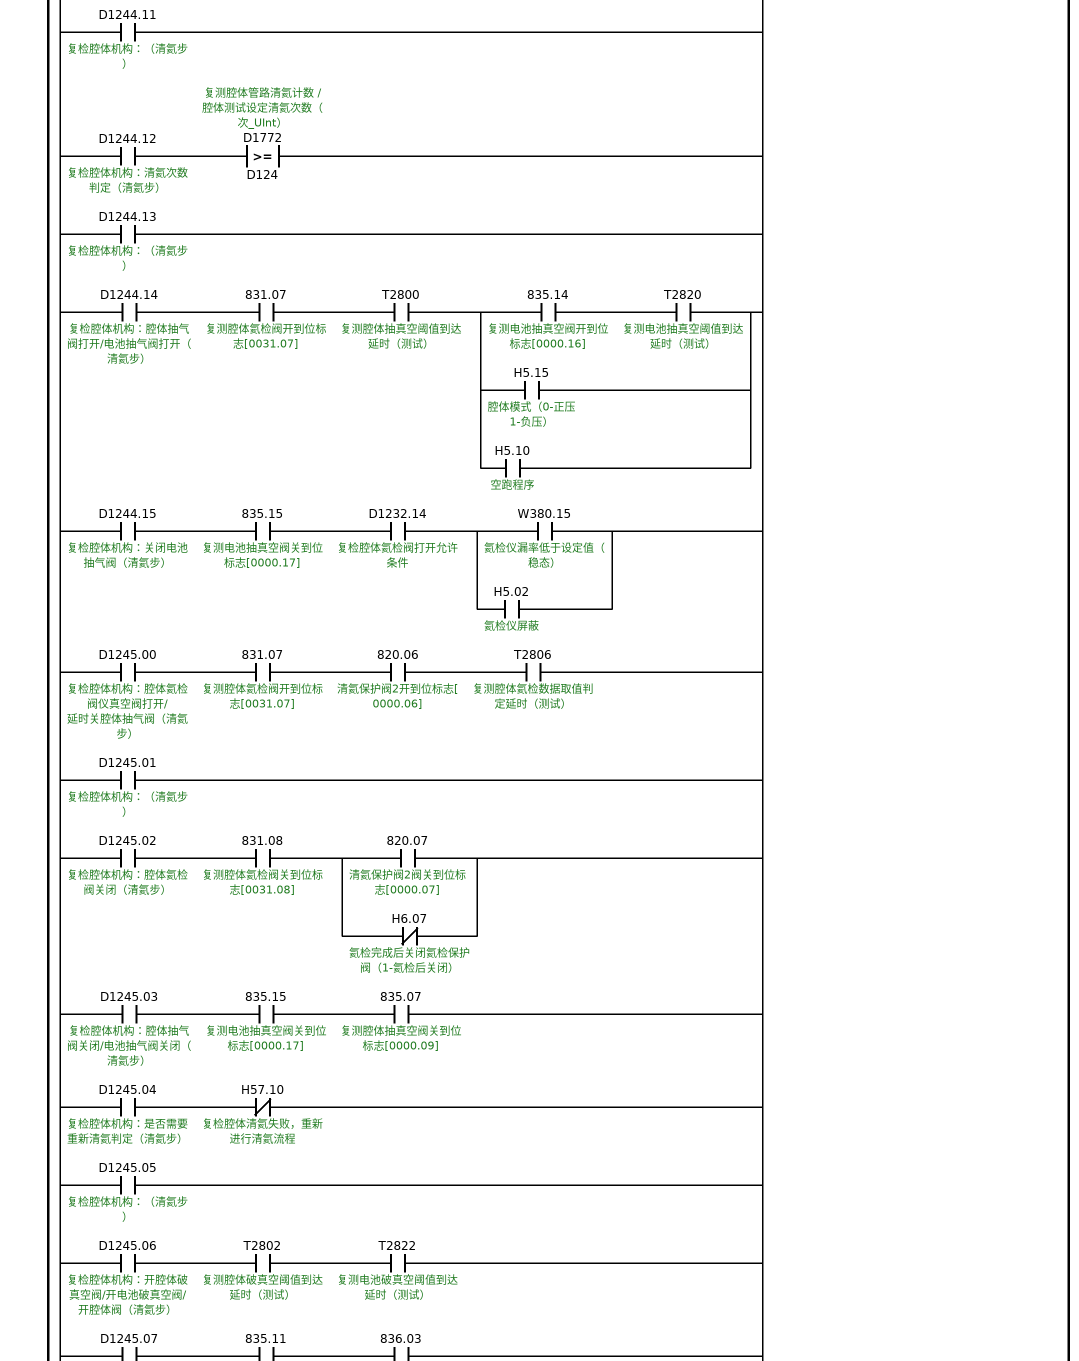

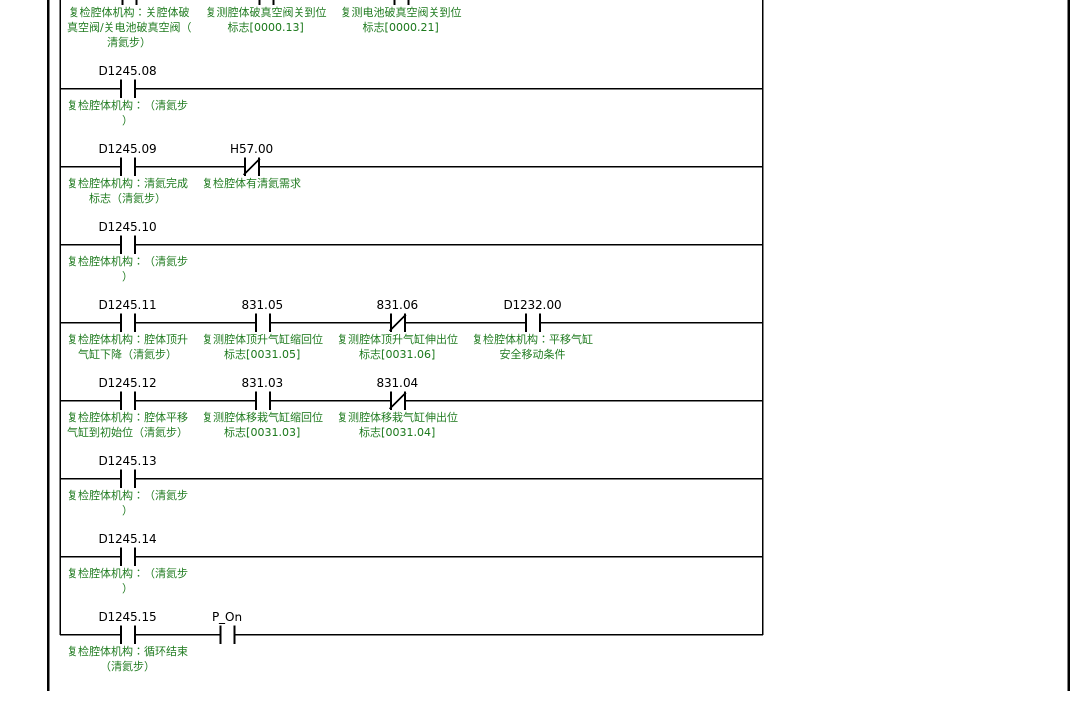
; rung 15
LD D1244.00  ; 复检腔体机构：自动开始（清氦步）
AND T1656  ; 复检腔体机构：开始运行延时（清氦步）
LD D1244.01  ; 复检腔体机构：平移气缸到氦检位/数据初始化（清氦步）
ANDNOT 831.03  ; 复测腔体移栽气缸缩回位标志[0031.03]
AND 831.04  ; 复测腔体移栽气缸伸出位标志[0031.04]
AND T2840  ; 复测数据初始化延时（清氦）
ORLD
LD D1244.02  ; 复检腔体机构：腔体顶升气缸上升（清氦步）
ANDNOT 831.05  ; 复测腔体顶升气缸缩回位标志[0031.05]
AND 831.06  ; 复测腔体顶升气缸伸出位标志[0031.06]
ORLD
LD D1244.03  ; 复检腔体机构：氦检仪真空阀关闭（清氦步）
AND 820.07  ; 清氦保护阀2阀关到位标志[0000.07]
ORLD
LD D1244.04  ; 复检腔体机构：正压开腔体阀/负压关腔体阀/氦检阀打开  // 负压模式下，复测前的清氦不允许抽电池
AND D1232.15  ; 复检腔体机构：腔体抽气阀打开允许
AND 831.07  ; 复测腔体氦检阀开到位标志[0031.07]
AND D1232.14  ; 复检腔体氦检阀打开允许条件
ORLD
OR D1244.05  ; 复检腔体机构：（清氦步）
LD D1244.06  ; 复检腔体机构：腔体抽气阀打开/电池抽气阀打开（清氦步）
LD T2800  ; 复测腔体抽真空阈值到达延时（测试）
OR T2808  ; 复测腔体抽残气时间上限到达延时（测试）
ANDLD
LD 835.14  ; 复测电池抽真空阀开到位标志[0000.16]
AND T2820  ; 复测电池抽真空阈值到达延时（测试）
OR T2821  ; 复测电池抽真空时间上限到达延时（测试）
OR H5.15  ; 腔体模式（0-正压 1-负压）
OR H5.10  ; 空跑程序
ANDLD
ORLD
LD D1244.07  ; 复检腔体机构：腔体抽气阀关闭/电池抽气阀关闭（清氦步）
AND 820.09  ; 清氦抽真空阀2关到位标志[0000.09]
AND 835.07  ; 复测腔体抽真空阀关到位标志[0000.09]
AND 835.15  ; 复测电池抽真空阀关到位标志[0000.17]
ORLD
OR D1244.08  ; 复检腔体机构：（清氦步）
LD D1244.09  ; 复检腔体机构：氦检清洁阀打开/电池破真空阀打开（清氦步）
AND T2841  ; 复测清氦注氮时长（清氦）
LD T2822  ; 复测电池破真空阈值到达延时（测试）
LD T2823  ; 复测电池破真空时间上限到达延时（测试）
OR H5.15  ; 腔体模式（0-正压 1-负压）
OR H5.10  ; 空跑程序
ORLD
ANDLD
ORLD
LD D1244.10  ; 复检腔体机构：氦检清洁阀关闭/电池破真空阀关闭（清氦步）
AND 820.09  ; 清氦抽真空阀2关到位标志[0000.09]
AND 835.07  ; 复测腔体抽真空阀关到位标志[0000.09]
AND 836.03  ; 复测电池破真空阀关到位标志[0000.21]
ORLD
OR D1244.11  ; 复检腔体机构：（清氦步）
LD D1244.12  ; 复检腔体机构：清氦次数判定（清氦步）
AND>=(325) D1772 D124  ; 复测腔体管路清氦计数, 腔体测试设定清氦次数（次_UInt）
ORLD
OR D1244.13  ; 复检腔体机构：（清氦步）
LD D1244.14  ; 复检腔体机构：腔体抽气阀打开/电池抽气阀打开（清氦步）
AND 831.07  ; 复测腔体氦检阀开到位标志[0031.07]
AND T2800  ; 复测腔体抽真空阈值到达延时（测试）
LD 835.14  ; 复测电池抽真空阀开到位标志[0000.16]
AND T2820  ; 复测电池抽真空阈值到达延时（测试）
OR H5.15  ; 腔体模式（0-正压 1-负压）
OR H5.10  ; 空跑程序
ANDLD
ORLD
LD D1244.15  ; 复检腔体机构：关闭电池抽气阀（清氦步）
AND 835.15  ; 复测电池抽真空阀关到位标志[0000.17]
AND D1232.14  ; 复检腔体氦检阀打开允许条件
LD W380.15  ; 氦检仪漏率低于设定值（稳态）
OR H5.02  ; 氦检仪屏蔽
ANDLD
ORLD
LD D1245.00  ; 复检腔体机构：腔体氦检阀仪真空阀打开/延时关腔体抽气阀（清氦步）
AND 831.07  ; 复测腔体氦检阀开到位标志[0031.07]
AND 820.06  ; 清氦保护阀2开到位标志[0000.06]
AND T2806  ; 复测腔体氦检数据取值判定延时（测试）
ORLD
OR D1245.01  ; 复检腔体机构：（清氦步）
LD D1245.02  ; 复检腔体机构：腔体氦检阀关闭（清氦步）
AND 831.08  ; 复测腔体氦检阀关到位标志[0031.08]
LD 820.07  ; 清氦保护阀2阀关到位标志[0000.07]
ORNOT H6.07  ; 氦检完成后关闭氦检保护阀（1-氦检后关闭）
ANDLD
ORLD
LD D1245.03  ; 复检腔体机构：腔体抽气阀关闭/电池抽气阀关闭（清氦步）
AND 835.15  ; 复测电池抽真空阀关到位标志[0000.17]
AND 835.07  ; 复测腔体抽真空阀关到位标志[0000.09]
ORLD
LD D1245.04  ; 复检腔体机构：是否需要重新清氦判定（清氦步）
ANDNOT H57.10  ; 复检腔体清氦失败，重新进行清氦流程  // 清氦失败，重新进行清氦
ORLD
OR D1245.05  ; 复检腔体机构：（清氦步）
LD D1245.06  ; 复检腔体机构：开腔体破真空阀/开电池破真空阀/开腔体阀（清氦步）
AND T2802  ; 复测腔体破真空阈值到达延时（测试）
AND T2822  ; 复测电池破真空阈值到达延时（测试）
ORLD
LD D1245.07  ; 复检腔体机构：关腔体破真空阀/关电池破真空阀（清氦步）
AND 835.11  ; 复测腔体破真空阀关到位标志[0000.13]
AND 836.03  ; 复测电池破真空阀关到位标志[0000.21]
ORLD
OR D1245.08  ; 复检腔体机构：（清氦步）
LD D1245.09  ; 复检腔体机构：清氦完成标志（清氦步）
ANDNOT H57.00  ; 复检腔体有清氦需求
ORLD
OR D1245.10  ; 复检腔体机构：（清氦步）
LD D1245.11  ; 复检腔体机构：腔体顶升气缸下降（清氦步）
AND 831.05  ; 复测腔体顶升气缸缩回位标志[0031.05]
ANDNOT 831.06  ; 复测腔体顶升气缸伸出位标志[0031.06]
AND D1232.00  ; 复检腔体机构：平移气缸安全移动条件
ORLD
LD D1245.12  ; 复检腔体机构：腔体平移气缸到初始位（清氦步）
AND 831.03  ; 复测腔体移栽气缸缩回位标志[0031.03]
ANDNOT 831.04  ; 复测腔体移栽气缸伸出位标志[0031.04]
ORLD
OR D1245.13  ; 复检腔体机构：（清氦步）
OR D1245.14  ; 复检腔体机构：（清氦步）
LD D1245.15  ; 复检腔体机构：循环结束（清氦步）
AND P_On
ORLD
AND D1234.03  ; 复检腔体机构：自动循环运行中（清氦步）
OUT D1235.05  ; 复检腔体机构：步进条件（清氦步）

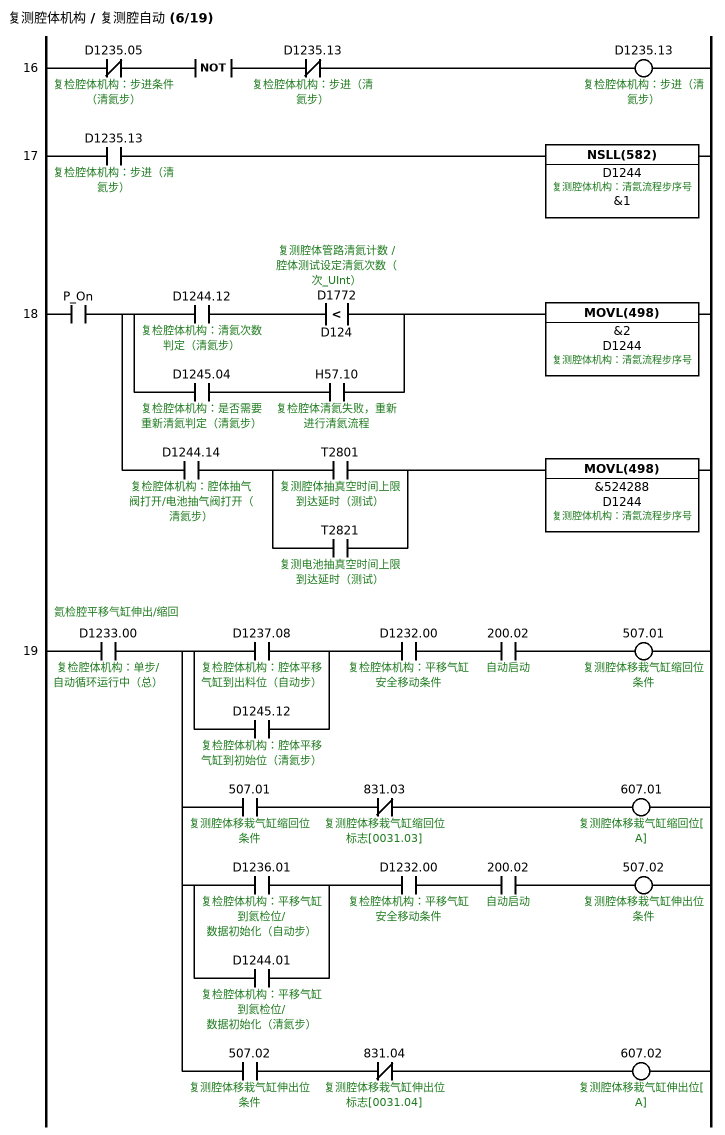
; rung 16
LDNOT D1235.05  ; 复检腔体机构：步进条件（清氦步）
NOT(520)
ANDNOT D1235.13  ; 复检腔体机构：步进（清氦步）
OUT D1235.13  ; 复检腔体机构：步进（清氦步）
; rung 17
LD D1235.13  ; 复检腔体机构：步进（清氦步）
NSLL(582) D1244 &1  ; 复测腔体机构：清氦流程步序号
; rung 18
LD P_On
OUT TR0
LD D1244.12  ; 复检腔体机构：清氦次数判定（清氦步）
AND<(310) D1772 D124  ; 复测腔体管路清氦计数, 腔体测试设定清氦次数（次_UInt）
LD D1245.04  ; 复检腔体机构：是否需要重新清氦判定（清氦步）
AND H57.10  ; 复检腔体清氦失败，重新进行清氦流程  // 清氦失败，重新进行清氦
ORLD
ANDLD
MOVL(498) &2 D1244  ; 复测腔体机构：清氦流程步序号
LD TR0
AND D1244.14  ; 复检腔体机构：腔体抽气阀打开/电池抽气阀打开（清氦步）
LD T2801  ; 复测腔体抽真空时间上限到达延时（测试）
OR T2821  ; 复测电池抽真空时间上限到达延时（测试）
ANDLD
MOVL(498) &524288 D1244  ; 复测腔体机构：清氦流程步序号  // 清氦过程腔体或电池抽气上限达到，均直接判定清氦完成，不进入氦检步序（跳转至D1075.03）
; rung 19: 氦检腔平移气缸伸出/缩回
LD D1233.00  ; 复检腔体机构：单步/自动循环运行中（总）
OUT TR0
LD D1237.08  ; 复检腔体机构：腔体平移气缸到出料位（自动步）
OR D1245.12  ; 复检腔体机构：腔体平移气缸到初始位（清氦步）
ANDLD
AND D1232.00  ; 复检腔体机构：平移气缸安全移动条件
AND 200.02  ; 自动启动
OUT 507.01  ; 复测腔体移栽气缸缩回位条件
LD TR0
AND 507.01  ; 复测腔体移栽气缸缩回位条件
ANDNOT 831.03  ; 复测腔体移栽气缸缩回位标志[0031.03]
OUT 607.01  ; 复测腔体移栽气缸缩回位[A]
LD TR0
LD D1236.01  ; 复检腔体机构：平移气缸到氦检位/数据初始化（自动步）
OR D1244.01  ; 复检腔体机构：平移气缸到氦检位/数据初始化（清氦步）
ANDLD
AND D1232.00  ; 复检腔体机构：平移气缸安全移动条件
AND 200.02  ; 自动启动
OUT 507.02  ; 复测腔体移栽气缸伸出位条件
LD TR0
AND 507.02  ; 复测腔体移栽气缸伸出位条件
ANDNOT 831.04  ; 复测腔体移栽气缸伸出位标志[0031.04]
OUT 607.02  ; 复测腔体移栽气缸伸出位[A]

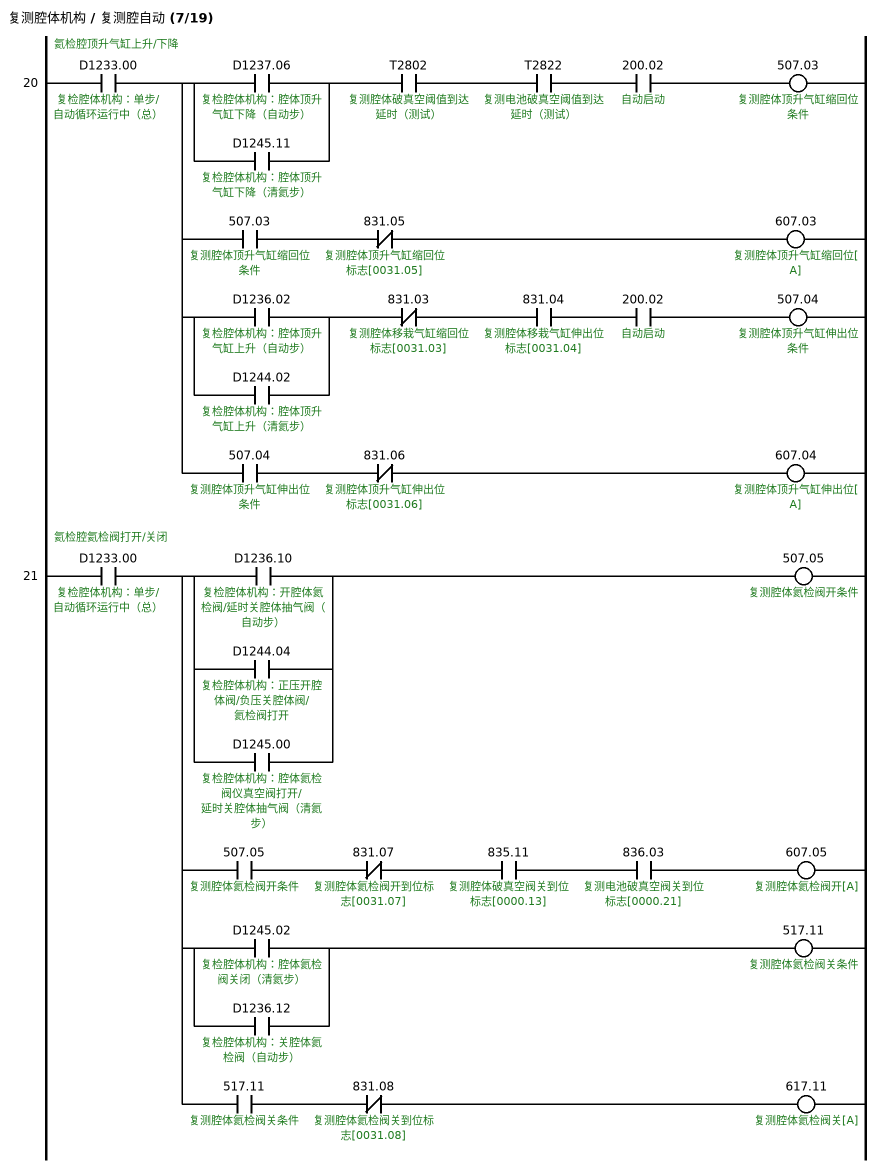
; rung 20: 氦检腔顶升气缸上升/下降
LD D1233.00  ; 复检腔体机构：单步/自动循环运行中（总）
OUT TR0
LD D1237.06  ; 复检腔体机构：腔体顶升气缸下降（自动步）
OR D1245.11  ; 复检腔体机构：腔体顶升气缸下降（清氦步）
ANDLD
AND T2802  ; 复测腔体破真空阈值到达延时（测试）
AND T2822  ; 复测电池破真空阈值到达延时（测试）
AND 200.02  ; 自动启动
OUT 507.03  ; 复测腔体顶升气缸缩回位条件
LD TR0
AND 507.03  ; 复测腔体顶升气缸缩回位条件
ANDNOT 831.05  ; 复测腔体顶升气缸缩回位标志[0031.05]
OUT 607.03  ; 复测腔体顶升气缸缩回位[A]
LD TR0
LD D1236.02  ; 复检腔体机构：腔体顶升气缸上升（自动步）
OR D1244.02  ; 复检腔体机构：腔体顶升气缸上升（清氦步）
ANDLD
ANDNOT 831.03  ; 复测腔体移栽气缸缩回位标志[0031.03]
AND 831.04  ; 复测腔体移栽气缸伸出位标志[0031.04]
AND 200.02  ; 自动启动
OUT 507.04  ; 复测腔体顶升气缸伸出位条件
LD TR0
AND 507.04  ; 复测腔体顶升气缸伸出位条件
ANDNOT 831.06  ; 复测腔体顶升气缸伸出位标志[0031.06]
OUT 607.04  ; 复测腔体顶升气缸伸出位[A]
; rung 21: 氦检腔氦检阀打开/关闭
LD D1233.00  ; 复检腔体机构：单步/自动循环运行中（总）
OUT TR0
LD D1236.10  ; 复检腔体机构：开腔体氦检阀/延时关腔体抽气阀（自动步）
OR D1244.04  ; 复检腔体机构：正压开腔体阀/负压关腔体阀/氦检阀打开
OR D1245.00  ; 复检腔体机构：腔体氦检阀仪真空阀打开/延时关腔体抽气阀（清氦步）
ANDLD
OUT 507.05  ; 复测腔体氦检阀开条件
LD TR0
AND 507.05  ; 复测腔体氦检阀开条件
ANDNOT 831.07  ; 复测腔体氦检阀开到位标志[0031.07]
AND 835.11  ; 复测腔体破真空阀关到位标志[0000.13]
AND 836.03  ; 复测电池破真空阀关到位标志[0000.21]
OUT 607.05  ; 复测腔体氦检阀开[A]
LD TR0
LD D1245.02  ; 复检腔体机构：腔体氦检阀关闭（清氦步）
OR D1236.12  ; 复检腔体机构：关腔体氦检阀（自动步）
ANDLD
OUT 517.11  ; 复测腔体氦检阀关条件
LD TR0
AND 517.11  ; 复测腔体氦检阀关条件
ANDNOT 831.08  ; 复测腔体氦检阀关到位标志[0031.08]
OUT 617.11  ; 复测腔体氦检阀关[A]

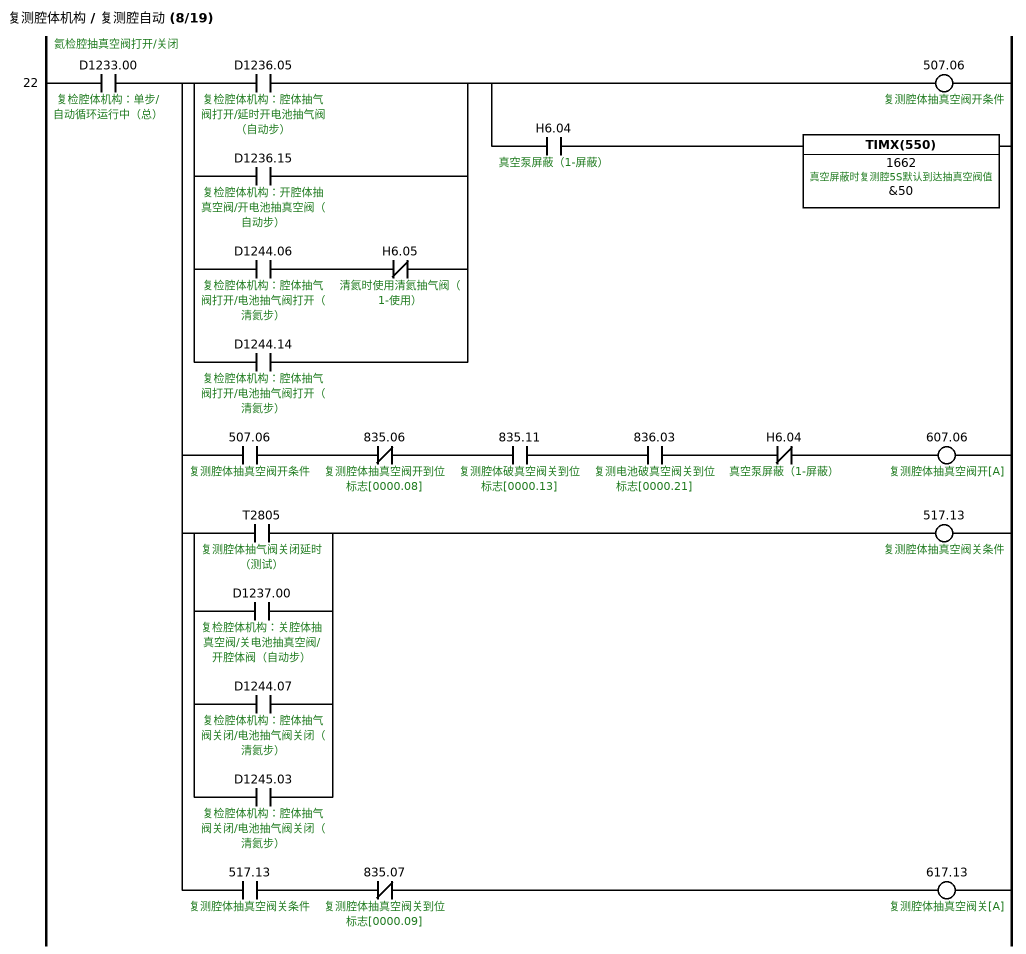
; rung 22: 氦检腔抽真空阀打开/关闭
LD D1233.00  ; 复检腔体机构：单步/自动循环运行中（总）
OUT TR0
LD D1236.05  ; 复检腔体机构：腔体抽气阀打开/延时开电池抽气阀（自动步）
OR D1236.15  ; 复检腔体机构：开腔体抽真空阀/开电池抽真空阀（自动步）
LD D1244.06  ; 复检腔体机构：腔体抽气阀打开/电池抽气阀打开（清氦步）
ANDNOT H6.05  ; 清氦时使用清氦抽气阀（1-使用）
ORLD
OR D1244.14  ; 复检腔体机构：腔体抽气阀打开/电池抽气阀打开（清氦步）
ANDLD
OUT 507.06  ; 复测腔体抽真空阀开条件
AND H6.04  ; 真空泵屏蔽（1-屏蔽）
TIMX(550) 1662 &50  ; 真空屏蔽时复测腔5S默认到达抽真空阀值
LD TR0
AND 507.06  ; 复测腔体抽真空阀开条件
ANDNOT 835.06  ; 复测腔体抽真空阀开到位标志[0000.08]
AND 835.11  ; 复测腔体破真空阀关到位标志[0000.13]
AND 836.03  ; 复测电池破真空阀关到位标志[0000.21]
ANDNOT H6.04  ; 真空泵屏蔽（1-屏蔽）
OUT 607.06  ; 复测腔体抽真空阀开[A]
LD TR0
LD T2805  ; 复测腔体抽气阀关闭延时（测试）
OR D1237.00  ; 复检腔体机构：关腔体抽真空阀/关电池抽真空阀/开腔体阀（自动步）
OR D1244.07  ; 复检腔体机构：腔体抽气阀关闭/电池抽气阀关闭（清氦步）
OR D1245.03  ; 复检腔体机构：腔体抽气阀关闭/电池抽气阀关闭（清氦步）
ANDLD
OUT 517.13  ; 复测腔体抽真空阀关条件
LD TR0
AND 517.13  ; 复测腔体抽真空阀关条件
ANDNOT 835.07  ; 复测腔体抽真空阀关到位标志[0000.09]
OUT 617.13  ; 复测腔体抽真空阀关[A]

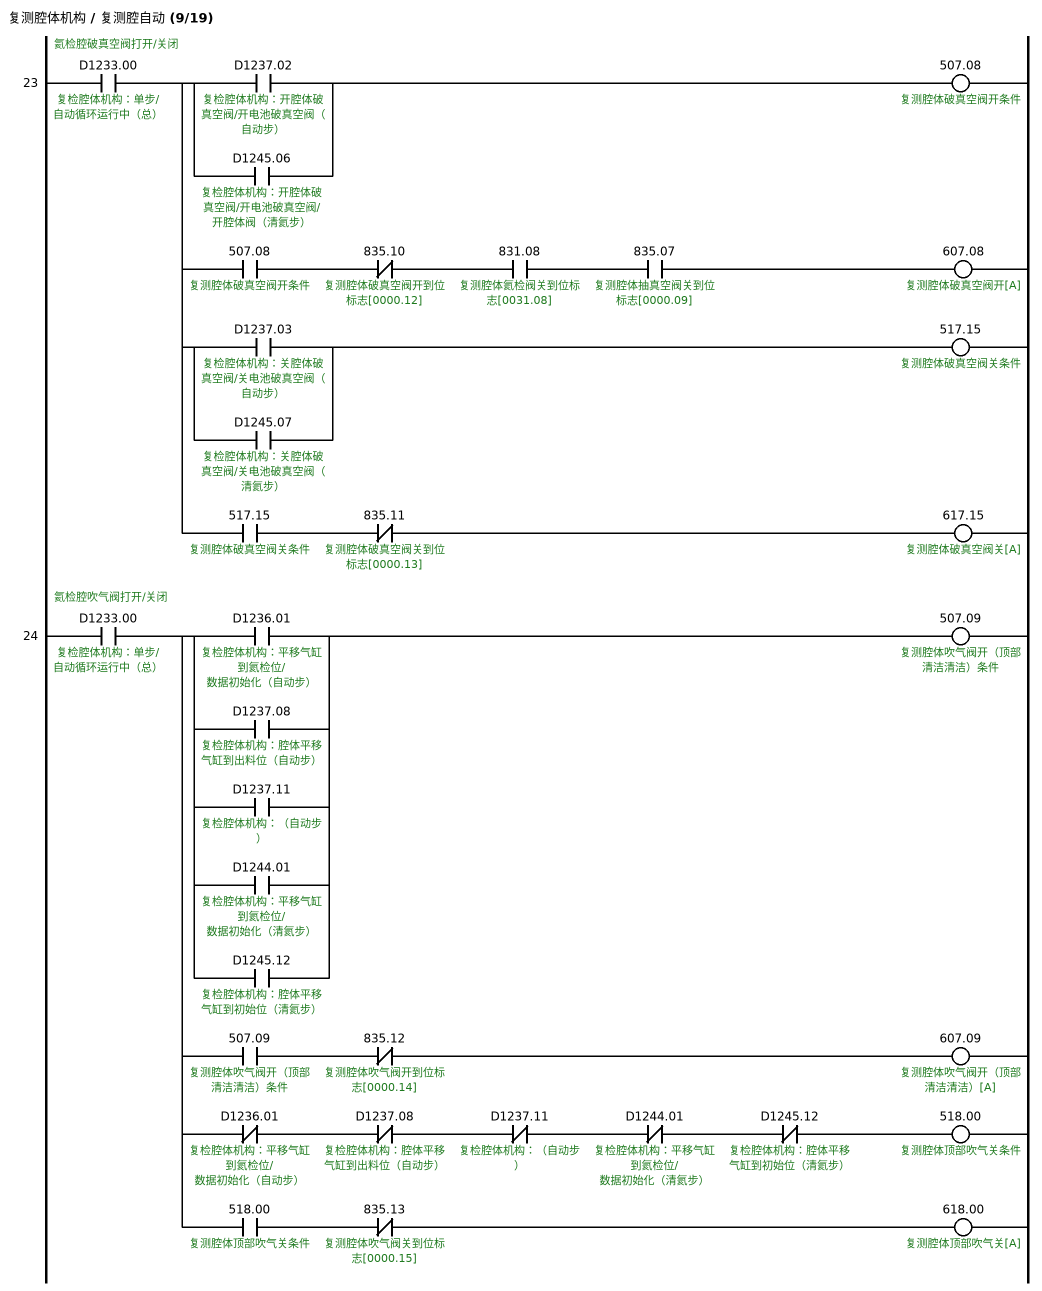
; rung 23: 氦检腔破真空阀打开/关闭
LD D1233.00  ; 复检腔体机构：单步/自动循环运行中（总）
OUT TR0
LD D1237.02  ; 复检腔体机构：开腔体破真空阀/开电池破真空阀（自动步）
OR D1245.06  ; 复检腔体机构：开腔体破真空阀/开电池破真空阀/开腔体阀（清氦步）
ANDLD
OUT 507.08  ; 复测腔体破真空阀开条件
LD TR0
AND 507.08  ; 复测腔体破真空阀开条件
ANDNOT 835.10  ; 复测腔体破真空阀开到位标志[0000.12]
AND 831.08  ; 复测腔体氦检阀关到位标志[0031.08]
AND 835.07  ; 复测腔体抽真空阀关到位标志[0000.09]
OUT 607.08  ; 复测腔体破真空阀开[A]
LD TR0
LD D1237.03  ; 复检腔体机构：关腔体破真空阀/关电池破真空阀（自动步）
OR D1245.07  ; 复检腔体机构：关腔体破真空阀/关电池破真空阀（清氦步）
ANDLD
OUT 517.15  ; 复测腔体破真空阀关条件
LD TR0
AND 517.15  ; 复测腔体破真空阀关条件
ANDNOT 835.11  ; 复测腔体破真空阀关到位标志[0000.13]
OUT 617.15  ; 复测腔体破真空阀关[A]
; rung 24: 氦检腔吹气阀打开/关闭
LD D1233.00  ; 复检腔体机构：单步/自动循环运行中（总）
OUT TR0
LD D1236.01  ; 复检腔体机构：平移气缸到氦检位/数据初始化（自动步）
OR D1237.08  ; 复检腔体机构：腔体平移气缸到出料位（自动步）
OR D1237.11  ; 复检腔体机构：（自动步）
OR D1244.01  ; 复检腔体机构：平移气缸到氦检位/数据初始化（清氦步）
OR D1245.12  ; 复检腔体机构：腔体平移气缸到初始位（清氦步）
ANDLD
OUT 507.09  ; 复测腔体吹气阀开（顶部清洁清洁）条件
LD TR0
AND 507.09  ; 复测腔体吹气阀开（顶部清洁清洁）条件
ANDNOT 835.12  ; 复测腔体吹气阀开到位标志[0000.14]
OUT 607.09  ; 复测腔体吹气阀开（顶部清洁清洁）[A]
LD TR0
ANDNOT D1236.01  ; 复检腔体机构：平移气缸到氦检位/数据初始化（自动步）
ANDNOT D1237.08  ; 复检腔体机构：腔体平移气缸到出料位（自动步）
ANDNOT D1237.11  ; 复检腔体机构：（自动步）
ANDNOT D1244.01  ; 复检腔体机构：平移气缸到氦检位/数据初始化（清氦步）
ANDNOT D1245.12  ; 复检腔体机构：腔体平移气缸到初始位（清氦步）
OUT 518.00  ; 复测腔体顶部吹气关条件
LD TR0
AND 518.00  ; 复测腔体顶部吹气关条件
ANDNOT 835.13  ; 复测腔体吹气阀关到位标志[0000.15]
OUT 618.00  ; 复测腔体顶部吹气关[A]

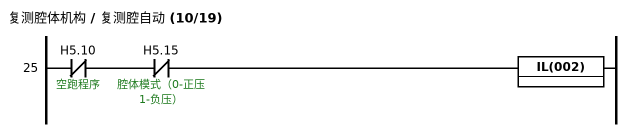
; rung 25
LDNOT H5.10  ; 空跑程序
ANDNOT H5.15  ; 腔体模式（0-正压 1-负压）
IL(002)

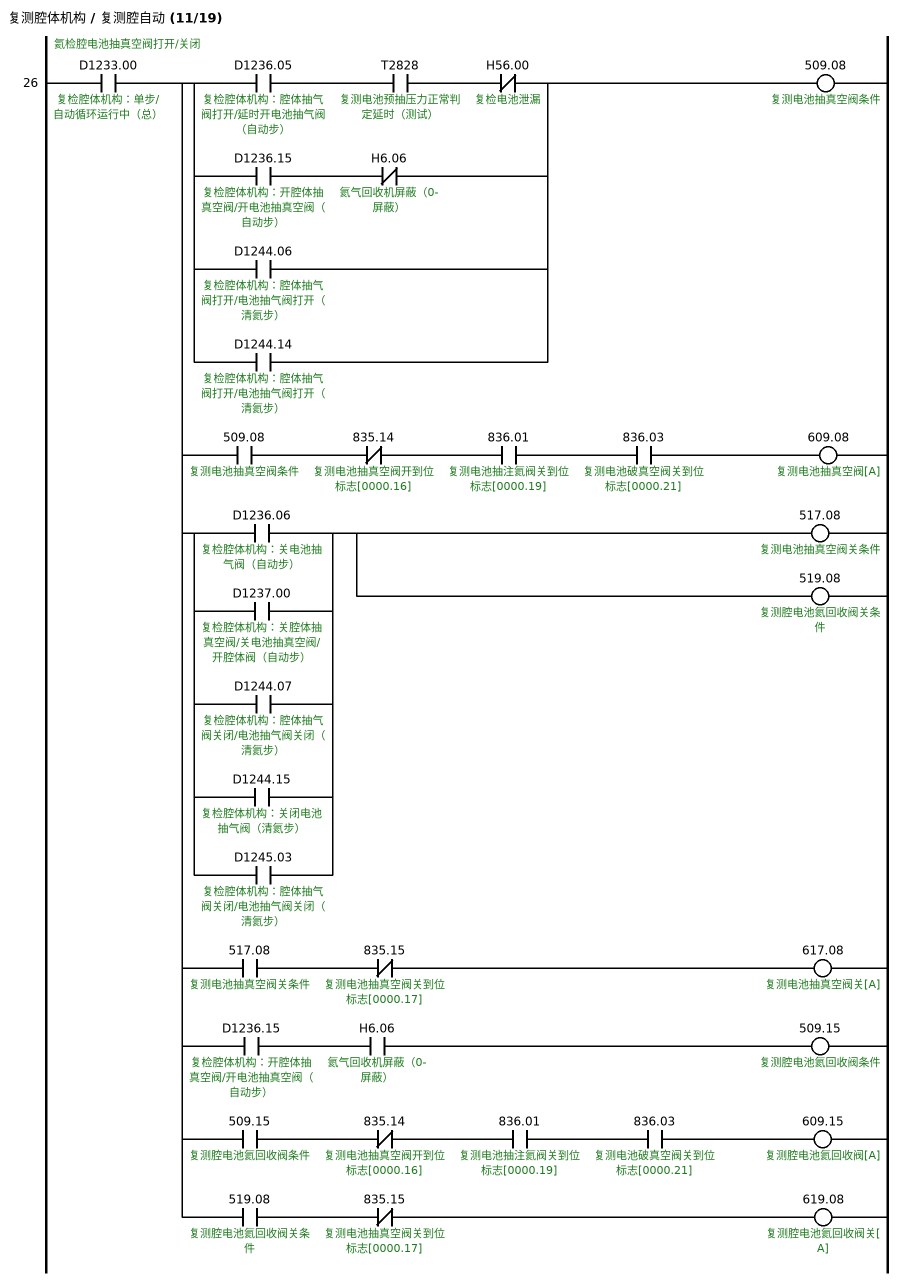
; rung 26: 氦检腔电池抽真空阀打开/关闭
LD D1233.00  ; 复检腔体机构：单步/自动循环运行中（总）
OUT TR0
LD D1236.05  ; 复检腔体机构：腔体抽气阀打开/延时开电池抽气阀（自动步）
AND T2828  ; 复测电池预抽压力正常判定延时（测试）
ANDNOT H56.00  ; 复检电池泄漏
LD D1236.15  ; 复检腔体机构：开腔体抽真空阀/开电池抽真空阀（自动步）
ANDNOT H6.06  ; 氦气回收机屏蔽（0-屏蔽）
ORLD
OR D1244.06  ; 复检腔体机构：腔体抽气阀打开/电池抽气阀打开（清氦步）
OR D1244.14  ; 复检腔体机构：腔体抽气阀打开/电池抽气阀打开（清氦步）
ANDLD
OUT 509.08  ; 复测电池抽真空阀条件
LD TR0
AND 509.08  ; 复测电池抽真空阀条件
ANDNOT 835.14  ; 复测电池抽真空阀开到位标志[0000.16]
AND 836.01  ; 复测电池抽注氦阀关到位标志[0000.19]
AND 836.03  ; 复测电池破真空阀关到位标志[0000.21]
OUT 609.08  ; 复测电池抽真空阀[A]
LD TR0
LD D1236.06  ; 复检腔体机构：关电池抽气阀（自动步）
OR D1237.00  ; 复检腔体机构：关腔体抽真空阀/关电池抽真空阀/开腔体阀（自动步）
OR D1244.07  ; 复检腔体机构：腔体抽气阀关闭/电池抽气阀关闭（清氦步）
OR D1244.15  ; 复检腔体机构：关闭电池抽气阀（清氦步）
OR D1245.03  ; 复检腔体机构：腔体抽气阀关闭/电池抽气阀关闭（清氦步）
ANDLD
OUT 517.08  ; 复测电池抽真空阀关条件
OUT 519.08  ; 复测腔电池氦回收阀关条件
LD TR0
AND 517.08  ; 复测电池抽真空阀关条件
ANDNOT 835.15  ; 复测电池抽真空阀关到位标志[0000.17]
OUT 617.08  ; 复测电池抽真空阀关[A]
LD TR0
AND D1236.15  ; 复检腔体机构：开腔体抽真空阀/开电池抽真空阀（自动步）
AND H6.06  ; 氦气回收机屏蔽（0-屏蔽）
OUT 509.15  ; 复测腔电池氦回收阀条件
LD TR0
AND 509.15  ; 复测腔电池氦回收阀条件
ANDNOT 835.14  ; 复测电池抽真空阀开到位标志[0000.16]
AND 836.01  ; 复测电池抽注氦阀关到位标志[0000.19]
AND 836.03  ; 复测电池破真空阀关到位标志[0000.21]
OUT 609.15  ; 复测腔电池氦回收阀[A]
LD TR0
AND 519.08  ; 复测腔电池氦回收阀关条件
ANDNOT 835.15  ; 复测电池抽真空阀关到位标志[0000.17]
OUT 619.08  ; 复测腔电池氦回收阀关[A]

